	88:
		BCGapMove:=FALSE;
		BCGapState:=0;
		BCGapBusy:=FALSE;
		BCGapDone:=TRUE;
		Error:=FALSE;
		ErrorID:=0;
		LeftTop_MC_MoveAbsolute.Execute:=FALSE;
		LeftBottom_MC_MoveAbsolute.Execute:=FALSE;
		RightTopLin_MC_MoveAbsolute.Execute:=FALSE;
		RightBottomLin_MC_MoveAbsolute.Execute:=FALSE;
		LeftIn_MC_MoveAbsolute.Execute:=FALSE;
		LeftOut_MC_MoveAbsolute.Execute:=FALSE;
		RightInLin_MC_MoveAbsolute.Execute:=FALSE;
		RightOutLin_MC_MoveAbsolute.Execute:=FALSE;
		fb_ton_BC.IN:=FALSE;
	89:
		BCGapMove:=FALSE;
		BCGapState:=0;
		BCGapBusy:=FALSE;
		BCGapDone:=FALSE;
		Error:=FALSE;
		ErrorID:=0;
		LeftTop_MC_MoveAbsolute.Execute:=FALSE;
		LeftBottom_MC_MoveAbsolute.Execute:=FALSE;
		RightTopLin_MC_MoveAbsolute.Execute:=FALSE;
		RightBottomLin_MC_MoveAbsolute.Execute:=FALSE;
		LeftIn_MC_MoveAbsolute.Execute:=FALSE;
		LeftOut_MC_MoveAbsolute.Execute:=FALSE;
		RightInLin_MC_MoveAbsolute.Execute:=FALSE;
		RightOutLin_MC_MoveAbsolute.Execute:=FALSE;
		fb_ton_BC.IN:=FALSE;
	99:
		BCGapMove:=FALSE;
		BCGapState:=99;
		BCGapBusy:=FALSE;
		BCGapDone:=FALSE;
		Error:=TRUE;
		LeftTop_MC_MoveAbsolute.Execute:=FALSE;
		LeftBottom_MC_MoveAbsolute.Execute:=FALSE;
		RightTopLin_MC_MoveAbsolute.Execute:=FALSE;
		RightBottomLin_MC_MoveAbsolute.Execute:=FALSE;
		LeftIn_MC_MoveAbsolute.Execute:=FALSE;
		LeftOut_MC_MoveAbsolute.Execute:=FALSE;
		RightInLin_MC_MoveAbsolute.Execute:=FALSE;
		RightOutLin_MC_MoveAbsolute.Execute:=FALSE;
		fb_ton_BC.IN:=FALSE;
	-100:
		FB_PlcEmergencyStop();
		BCGapMove:=FALSE;
		BCGapState:=-100;
		BCGapBusy:=FALSE;
		BCGapDone:=FALSE;
		Error:=TRUE;
		LeftTop_MC_MoveAbsolute.Execute:=FALSE;
		LeftBottom_MC_MoveAbsolute.Execute:=FALSE;
		RightTopLin_MC_MoveAbsolute.Execute:=FALSE;
		RightBottomLin_MC_MoveAbsolute.Execute:=FALSE;
		LeftIn_MC_MoveAbsolute.Execute:=FALSE;
		LeftOut_MC_MoveAbsolute.Execute:=FALSE;
		RightInLin_MC_MoveAbsolute.Execute:=FALSE;
		RightOutLin_MC_MoveAbsolute.Execute:=FALSE;
		fb_ton_BC.IN:=FALSE;
END_CASE
END_IF
END_ACTION

ACTION A_BottomMove:
IF BottomMove THEN
BottomBusy:=TRUE;
BottomDone:=FALSE;
fb_ton2(PT:=t#80s);(*2mm/s max spees,120mmÐÐ³Ì£¬60sÄÚ×ßÍê*)
A_MoveMC();
CASE BottomState OF

	0:
		IF  LeftBottom_MC_MoveAbsolute.Error OR RightBottomLin_MC_MoveAbsolute.Error THEN		(*¼ì²éMC Error*)
			ErrorID:=2;
			BottomState:=99;
		END_IF
		BottomState:=1;

	1:
		LeftBottom_MC_MoveAbsolute.Position:=BottomPosition;
		LeftBottom_MC_MoveAbsolute.Velocity:=BottomVelocity;
		LeftBottom_MC_MoveAbsolute.Execute:=TRUE;
		RightBottomLin_MC_MoveAbsolute.Position:=BottomPosition;
		RightBottomLin_MC_MoveAbsolute.Velocity:=BottomVelocity;
		RightBottomLin_MC_MoveAbsolute.Execute:=TRUE;
		fb_ton2.IN:=TRUE;
		BottomState:=2;
	2:
		IF NOT LeftBottom_MC_MoveAbsolute.Done THEN		(*ÔË¶¯ÖÐ£¬¼ì²éDoneÐÅºÅ£¬Ã»ÓÐÔòÑ­»·£¬³¬Ê±±¨´í*)
			BottomState:=2;
		ELSIF LeftBottom_MC_MoveAbsolute.Done THEN		(*ÔË¶¯Íê³É£¬×ªÏÂÒ»²½*)
				BottomState:=88;
		END_IF
		(*½ÓÊÕµ½stopÐÅºÅÊ±£¬reset×´Ì¬*)
		IF BottomReset THEN
			BottomState:=89;
		END_IF

	88:
		BottomMove:=FALSE;
		BottomState:=0;
		BottomBusy:=FALSE;
		BottomDone:=TRUE;
		Error:=FALSE;
		ErrorID:=0;
		LeftBottom_MC_MoveAbsolute.Execute:=FALSE;
		RightBottomLin_MC_MoveAbsolute.Execute:=FALSE;
		fb_ton2.IN:=FALSE;
	89:
		BottomMove:=FALSE;
		BottomState:=0;
		BottomBusy:=FALSE;
		BottomDone:=FALSE;
		Error:=FALSE;
		ErrorID:=0;
		LeftBottom_MC_MoveAbsolute.Execute:=FALSE;
		RightBottomLin_MC_MoveAbsolute.Execute:=FALSE;
		fb_ton2.IN:=FALSE;
	99:
		BottomMove:=FALSE;
		BottomState:=99;
		BottomBusy:=FALSE;
		BottomDone:=FALSE;
		Error:=TRUE;
		LeftBottom_MC_MoveAbsolute.Execute:=FALSE;
		RightBottomLin_MC_MoveAbsolute.Execute:=FALSE;
		fb_ton2.IN:=FALSE;
	-100:
		FB_PlcEmergencyStop();
		BottomMove:=FALSE;
		BottomState:=-100;
		BottomBusy:=FALSE;
		BottomDone:=FALSE;
		Error:=TRUE;
		LeftBottom_MC_MoveAbsolute.Execute:=FALSE;
		RightBottomLin_MC_MoveAbsolute.Execute:=FALSE;
		fb_ton2.IN:=FALSE;
END_CASE
END_IF
END_ACTION

ACTION A_InMove:
IF InMove THEN
InBusy:=TRUE;
InDone:=FALSE;
fb_ton3(PT:=T#80S);(*2mm/s max spees,120mmÐÐ³Ì£¬60sÄÚ×ßÍê*)
A_MoveMC();
CASE InState OF
	0:
		IF LeftIn_MC_MoveAbsolute.Error OR RightInLin_MC_MoveAbsolute.Error THEN		(*¼ì²éMC Error*)
			ErrorID:=2;
			InState:=99;
		END_IF
		InState:=1;
	1:
		LeftIn_MC_MoveAbsolute.Position:=InPosition;
		LeftIn_MC_MoveAbsolute.Velocity:=InVelocity;
		LeftIn_MC_MoveAbsolute.Execute:=TRUE;
		RightInLin_MC_MoveAbsolute.Position:=InPosition;
		RightInLin_MC_MoveAbsolute.Velocity:=InVelocity;
		RightInLin_MC_MoveAbsolute.Execute:=TRUE;
		fb_ton3.IN:=TRUE;
		InState:=2;
	2:
		IF NOT LeftIn_MC_MoveAbsolute.Done OR NOT RightInLin_MC_MoveAbsolute.Done THEN		(*ÔË¶¯ÖÐ£¬¼ì²éDoneÐÅºÅ£¬Ã»ÓÐÔòÑ­»·£¬³¬Ê±±¨´í*)
			InState:=2;
		ELSIF LeftIn_MC_MoveAbsolute.Done AND RightInLin_MC_MoveAbsolute.Done THEN		(*ÔË¶¯Íê³É£¬×ªÏÂÒ»²½*)
				InState:=88;
		END_IF
		(*½ÓÊÕµ½sInÐÅºÅÊ±£¬reset×´Ì¬*)
		IF InReset THEN
			InState:=89;
		END_IF

	88:
		InMove:=FALSE;
		InState:=0;
		InBusy:=FALSE;
		InDone:=TRUE;
		Error:=FALSE;
		ErrorID:=0;
		LeftIn_MC_MoveAbsolute.Execute:=FALSE;
		RightInLin_MC_MoveAbsolute.Execute:=FALSE;
		fb_ton3.IN:=FALSE;
	89:
		InMove:=FALSE;
		InState:=0;
		InBusy:=FALSE;
		InDone:=FALSE;
		Error:=FALSE;
		ErrorID:=0;
		LeftIn_MC_MoveAbsolute.Execute:=FALSE;
		RightInLin_MC_MoveAbsolute.Execute:=FALSE;
		fb_ton3.IN:=FALSE;
	99:
		InMove:=FALSE;
		InState:=99;
		InBusy:=FALSE;
		InDone:=FALSE;
		Error:=TRUE;
		LeftIn_MC_MoveAbsolute.Execute:=FALSE;
		RightInLin_MC_MoveAbsolute.Execute:=FALSE;
		fb_ton3.IN:=FALSE;
	-100:
		FB_PlcEmergencyStop();
		InMove:=FALSE;
		InState:=-100;
		InBusy:=FALSE;
		InDone:=FALSE;
		Error:=TRUE;
		LeftIn_MC_MoveAbsolute.Execute:=FALSE;
		RightInLin_MC_MoveAbsolute.Execute:=FALSE;
		fb_ton3.IN:=FALSE;
END_CASE
END_IF
END_ACTION

ACTION A_LeftBottomMove:
IF LeftBottomMove THEN
LeftBottomBusy:=TRUE;
LeftBottomDone:=FALSE;
fb_ton_debug_3(PT:=t#10s);

A_MoveMC();
CASE LeftBottomState OF
	0:
		IF LeftBottom_MC_MoveAbsolute.Error THEN		(*¼ì²éMC Error*)
			ErrorID:=2;
			LeftBottomState:=99;
		ELSIF leftBottomLin.Status.NotMoving THEN	(*Öá¶¼´¦ÓÚÍ£Ö¹×´Ì¬Ê±£¬×ªÏÂÒ»²½*)
			LeftBottomState:=1;
		END_IF
	1:
		LeftBottom_MC_MoveAbsolute.Position:=LeftBottomPosition;
		LeftBottom_MC_MoveAbsolute.Velocity:=LeftBottomVelocity;
		LeftBottom_MC_MoveAbsolute.Execute:=TRUE;
		fb_ton_debug_3.IN:=TRUE;
		LeftBottomState:=2;
	2:
		IF NOT LeftBottom_MC_MoveAbsolute.Done THEN		(*ÔË¶¯ÖÐ£¬¼ì²éDoneÐÅºÅ£¬Ã»ÓÐÔòÑ­»·£¬³¬Ê±±¨´í*)
			LeftBottomState:=2;
		ELSIF LeftBottom_MC_MoveAbsolute.Done THEN		(*ÔË¶¯Íê³É£¬×ªÏÂÒ»²½*)
				LeftBottomState:=88;
		END_IF
		(*½ÓÊÕµ½stopÐÅºÅÊ±£¬reset×´Ì¬*)
		IF LeftBottomReset THEN
			LeftBottomState:=89;
		END_IF

	88:
		LeftBottomMove:=FALSE;
		LeftBottomState:=0;
		LeftBottomBusy:=FALSE;
		LeftBottomDone:=TRUE;
		Error:=FALSE;
		ErrorID:=0;
		LeftBottom_MC_MoveAbsolute.Execute:=FALSE;
		fb_ton_debug_3.IN:=FALSE;
	89:
		LeftBottomMove:=FALSE;
		LeftBottomState:=0;
		LeftBottomBusy:=FALSE;
		LeftBottomDone:=FALSE;
		Error:=FALSE;
		ErrorID:=0;
		LeftBottom_MC_MoveAbsolute.Execute:=FALSE;
		fb_ton_debug_3.IN:=FALSE;
	99:
		LeftBottomMove:=FALSE;
		LeftBottomState:=99;
		LeftBottomBusy:=FALSE;
		LeftBottomDone:=FALSE;
		Error:=TRUE;
		LeftBottom_MC_MoveAbsolute.Execute:=FALSE;
		fb_ton_debug_3.IN:=FALSE;
	-100:
		FB_PlcEmergencyStop();
		LeftBottomMove:=FALSE;
		LeftBottomState:=-100;
		LeftBottomBusy:=FALSE;
		LeftBottomDone:=FALSE;
		Error:=TRUE;
		LeftBottom_MC_MoveAbsolute.Execute:=FALSE;
		fb_ton_debug_3.IN:=FALSE;
END_CASE
END_IF
END_ACTION

ACTION A_LeftInMove:
IF LeftInMove THEN
LeftInBusy:=TRUE;
LeftInDone:=FALSE;
fb_ton_debug_5(PT:=T#10S);

A_MoveMC();
CASE LeftInState OF
	0:
		IF LeftIn_MC_MoveAbsolute.Error THEN		(*¼ì²éMC Error*)
			ErrorID:=2;
			LeftInState:=99;
		ELSIF leftInLin.Status.NotMoving THEN	(*Öá¶¼´¦ÓÚÍ£Ö¹×´Ì¬Ê±£¬×ªÏÂÒ»²½*)
			LeftInState:=1;
		END_IF
	1:
		LeftIn_MC_MoveAbsolute.Position:=LeftInPosition;
		LeftIn_MC_MoveAbsolute.Velocity:=LeftInVelocity;
		LeftIn_MC_MoveAbsolute.Execute:=TRUE;
		fb_ton_debug_5.IN:=TRUE;
		LeftInState:=2;
	2:
		IF NOT LeftIn_MC_MoveAbsolute.Done THEN		(*ÔË¶¯ÖÐ£¬¼ì²éDoneÐÅºÅ£¬Ã»ÓÐÔòÑ­»·£¬³¬Ê±±¨´í*)
			LeftInState:=2;
		ELSIF LeftIn_MC_MoveAbsolute.Done THEN		(*ÔË¶¯Íê³É£¬×ªÏÂÒ»²½*)
				LeftInState:=88;
		END_IF
		(*½ÓÊÕµ½stopÐÅºÅÊ±£¬reset×´Ì¬*)
		IF LeftInReset THEN
			LeftInState:=89;
		END_IF

	88:
		LeftInMove:=FALSE;
		LeftInState:=0;
		LeftInBusy:=FALSE;
		LeftInDone:=TRUE;
		Error:=FALSE;
		ErrorID:=0;
		LeftIn_MC_MoveAbsolute.Execute:=FALSE;
		fb_ton_debug_5.IN:=FALSE;
	89:
		LeftInMove:=FALSE;
		LeftInState:=0;
		LeftInBusy:=FALSE;
		LeftInDone:=FALSE;
		Error:=FALSE;
		ErrorID:=0;
		LeftIn_MC_MoveAbsolute.Execute:=FALSE;
		fb_ton_debug_5.IN:=FALSE;
	99:
		LeftInMove:=FALSE;
		LeftInState:=99;
		LeftInBusy:=FALSE;
		LeftInDone:=FALSE;
		Error:=TRUE;
		LeftIn_MC_MoveAbsolute.Execute:=FALSE;
		fb_ton_debug_5.IN:=FALSE;
	-100:
		FB_PlcEmergencyStop();
		LeftInMove:=FALSE;
		LeftInState:=-100;
		LeftInBusy:=FALSE;
		LeftInDone:=FALSE;
		Error:=TRUE;
		LeftIn_MC_MoveAbsolute.Execute:=FALSE;
		fb_ton_debug_5.IN:=FALSE;
END_CASE
END_IF
END_ACTION

ACTION A_LeftOutMove:
IF LeftOutMove THEN
LeftOutBusy:=TRUE;
LeftOutDone:=FALSE;
fb_ton_debug_7(PT:=t#10s);

A_MoveMC();
CASE LeftOutState OF
	0:
		IF LeftOut_MC_MoveAbsolute.Error THEN		(*¼ì²éMC Error*)
			ErrorID:=2;
			LeftOutState:=99;
		ELSIF leftOutLin.Status.NotMoving THEN	(*Öá¶¼´¦ÓÚÍ£Ö¹×´Ì¬Ê±£¬×ªÏÂÒ»²½*)
			LeftOutState:=1;
		END_IF
	1:
		LeftOut_MC_MoveAbsolute.Position:=LeftOutPosition;
		LeftOut_MC_MoveAbsolute.Velocity:=LeftOutVelocity;
		LeftOut_MC_MoveAbsolute.Execute:=TRUE;
		fb_ton_debug_7.IN:=TRUE;
		LeftOutState:=2;
	2:
		IF NOT LeftOut_MC_MoveAbsolute.Done THEN		(*ÔË¶¯ÖÐ£¬¼ì²éDoneÐÅºÅ£¬Ã»ÓÐÔòÑ­»·£¬³¬Ê±±¨´í*)
			LeftOutState:=2;
		ELSIF LeftOut_MC_MoveAbsolute.Done THEN		(*ÔË¶¯Íê³É£¬×ªÏÂÒ»²½*)
				LeftOutState:=88;
		END_IF
		(*½ÓÊÕµ½stopÐÅºÅÊ±£¬reset×´Ì¬*)
		IF LeftOutReset THEN
			LeftOutState:=89;
		END_IF

	88:
		LeftOutMove:=FALSE;
		LeftOutState:=0;
		LeftOutBusy:=FALSE;
		LeftOutDone:=TRUE;
		Error:=FALSE;
		ErrorID:=0;
		LeftOut_MC_MoveAbsolute.Execute:=FALSE;
		fb_ton_debug_7.IN:=FALSE;
	89:
		LeftOutMove:=FALSE;
		LeftOutState:=0;
		LeftOutBusy:=FALSE;
		LeftOutDone:=FALSE;
		Error:=FALSE;
		ErrorID:=0;
		LeftOut_MC_MoveAbsolute.Execute:=FALSE;
		fb_ton_debug_7.IN:=FALSE;
	99:
		LeftOutMove:=FALSE;
		LeftOutState:=99;
		LeftOutBusy:=FALSE;
		LeftOutDone:=FALSE;
		Error:=TRUE;
		LeftOut_MC_MoveAbsolute.Execute:=FALSE;
		fb_ton_debug_7.IN:=FALSE;
	-100:
		FB_PlcEmergencyStop();
		LeftOutMove:=FALSE;
		LeftOutState:=-100;
		LeftOutBusy:=FALSE;
		LeftOutDone:=FALSE;
		Error:=TRUE;
		LeftOut_MC_MoveAbsolute.Execute:=FALSE;
		fb_ton_debug_7.IN:=FALSE;
END_CASE
END_IF
END_ACTION

ACTION A_LeftTopMove:
IF LeftTopMove THEN
LeftTopBusy:=TRUE;
LeftTopDone:=FALSE;
fb_ton_debug_1(PT:=t#10s);

A_MoveMC();
CASE LeftTopState OF
	0:
		IF LeftTop_MC_MoveAbsolute.Error THEN		(*¼ì²éMC Error*)
			ErrorID:=2;
			LeftTopState:=99;
		ELSIF leftTopLin.Status.NotMoving THEN	(*Öá¶¼´¦ÓÚÍ£Ö¹×´Ì¬Ê±£¬×ªÏÂÒ»²½*)
			LeftTopState:=1;
		END_IF
	1:
		LeftTop_MC_MoveAbsolute.Position:=LeftTopPosition;
		LeftTop_MC_MoveAbsolute.Velocity:=LeftTopVelocity;
		LeftTop_MC_MoveAbsolute.Execute:=TRUE;
		fb_ton_debug_1.IN:=TRUE;
		LeftTopState:=2;
	2:
		IF NOT LeftTop_MC_MoveAbsolute.Done THEN		(*ÔË¶¯ÖÐ£¬¼ì²éDoneÐÅºÅ£¬Ã»ÓÐÔòÑ­»·£¬³¬Ê±±¨´í*)
			LeftTopState:=2;
		ELSIF LeftTop_MC_MoveAbsolute.Done THEN		(*ÔË¶¯Íê³É£¬×ªÏÂÒ»²½*)
				LeftTopState:=88;
		END_IF
		(*½ÓÊÕµ½stopÐÅºÅÊ±£¬reset×´Ì¬*)
		IF LeftTopReset THEN
			LeftTopState:=89;
		END_IF

	88:
		LeftTopMove:=FALSE;
		LeftTopState:=0;
		LeftTopBusy:=FALSE;
		LeftTopDone:=TRUE;
		Error:=FALSE;
		ErrorID:=0;
		LeftTop_MC_MoveAbsolute.Execute:=FALSE;
		fb_ton_debug_1.IN:=FALSE;
	89:
		LeftTopMove:=FALSE;
		LeftTopState:=0;
		LeftTopBusy:=FALSE;
		LeftTopDone:=FALSE;
		Error:=FALSE;
		ErrorID:=0;
		LeftTop_MC_MoveAbsolute.Execute:=FALSE;
		fb_ton_debug_1.IN:=FALSE;
	99:
		LeftTopMove:=FALSE;
		LeftTopState:=99;
		LeftTopBusy:=FALSE;
		LeftTopDone:=FALSE;
		Error:=TRUE;
		LeftTop_MC_MoveAbsolute.Execute:=FALSE;
		fb_ton_debug_1.IN:=FALSE;
	-100:
		FB_PlcEmergencyStop();
		LeftTopMove:=FALSE;
		LeftTopState:=-100;
		LeftTopBusy:=FALSE;
		LeftTopDone:=FALSE;
		Error:=TRUE;
		LeftTop_MC_MoveAbsolute.Execute:=FALSE;
		fb_ton_debug_1.IN:=FALSE;
END_CASE
END_IF
END_ACTION

ACTION A_MoveMC:
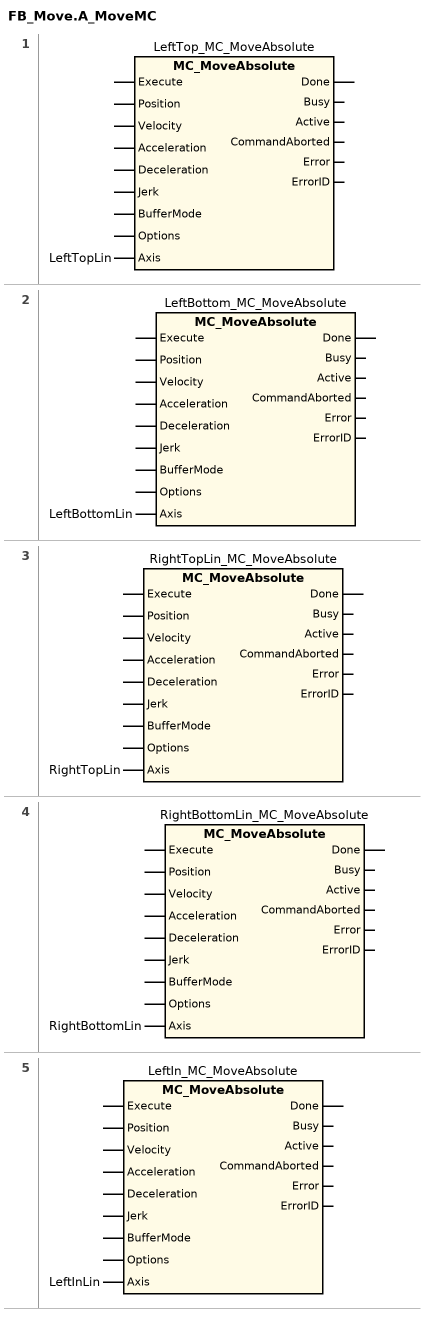
// NETWORK 1
LeftTop_MC_MoveAbsolute(Axis := LeftTopLin); // MC_MoveAbsolute

// NETWORK 2
LeftBottom_MC_MoveAbsolute(Axis := LeftBottomLin); // MC_MoveAbsolute

// NETWORK 3
RightTopLin_MC_MoveAbsolute(Axis := RightTopLin); // MC_MoveAbsolute

// NETWORK 4
RightBottomLin_MC_MoveAbsolute(Axis := RightBottomLin); // MC_MoveAbsolute

// NETWORK 5
LeftIn_MC_MoveAbsolute(Axis := LeftInLin); // MC_MoveAbsolute

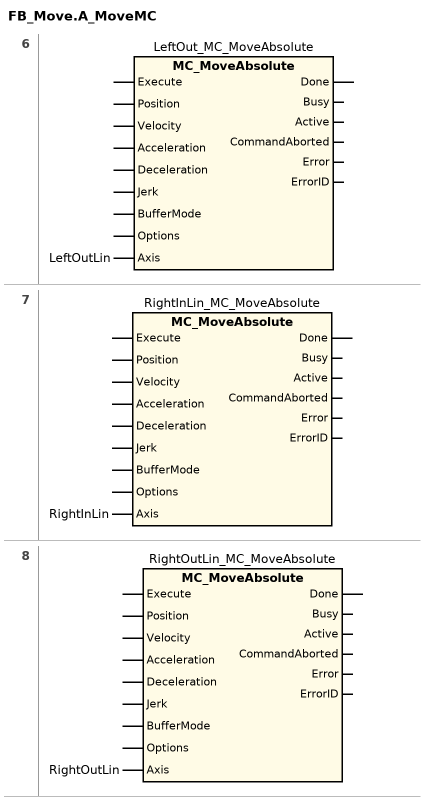
// NETWORK 6
LeftOut_MC_MoveAbsolute(Axis := LeftOutLin); // MC_MoveAbsolute

// NETWORK 7
RightInLin_MC_MoveAbsolute(Axis := RightInLin); // MC_MoveAbsolute

// NETWORK 8
RightOutLin_MC_MoveAbsolute(Axis := RightOutLin); // MC_MoveAbsolute
END_ACTION

ACTION A_OutMove:
IF OutMove THEN
OutBusy:=TRUE;
OutDone:=FALSE;
fb_ton4(PT:=T#80S);(*2mm/s max spees,120mmÐÐ³Ì£¬60sÄÚ×ßÍê*)
A_MoveMC();
CASE OutState OF

	0:
		IF  LeftOut_MC_MoveAbsolute.Error OR RightOutLin_MC_MoveAbsolute.Error THEN		(*¼ì²éMC Error*)
			ErrorID:=2;
			OutState:=99;
		END_IF
		OutState:=1;

	1:
		LeftOut_MC_MoveAbsolute.Position:=OutPosition;
		LeftOut_MC_MoveAbsolute.Velocity:=OutVelocity;
		LeftOut_MC_MoveAbsolute.Execute:=TRUE;
		RightOutLin_MC_MoveAbsolute.Position:=OutPosition;
		RightOutLin_MC_MoveAbsolute.Velocity:=OutVelocity;
		RightOutLin_MC_MoveAbsolute.Execute:=TRUE;
		fb_ton4.IN:=TRUE;
		OutState:=2;
	2:
		IF NOT LeftOut_MC_MoveAbsolute.Done THEN		(*ÔË¶¯ÖÐ£¬¼ì²éDoneÐÅºÅ£¬Ã»ÓÐÔòÑ­»·£¬³¬Ê±±¨´í*)
			OutState:=2;
		ELSIF LeftOut_MC_MoveAbsolute.Done THEN		(*ÔË¶¯Íê³É£¬×ªÏÂÒ»²½*)
				OutState:=88;
		END_IF
		(*½ÓÊÕµ½stopÐÅºÅÊ±£¬reset×´Ì¬*)
		IF OutReset THEN
			OutState:=89;
		END_IF

	88:
		OutMove:=FALSE;
		OutState:=0;
		OutBusy:=FALSE;
		OutDone:=TRUE;
		Error:=FALSE;
		ErrorID:=0;
		LeftOut_MC_MoveAbsolute.Execute:=FALSE;
		RightOutLin_MC_MoveAbsolute.Execute:=FALSE;
		fb_ton4.IN:=FALSE;
	89:
		OutMove:=FALSE;
		OutState:=0;
		OutBusy:=FALSE;
		OutDone:=FALSE;
		Error:=FALSE;
		ErrorID:=0;
		LeftOut_MC_MoveAbsolute.Execute:=FALSE;
		RightOutLin_MC_MoveAbsolute.Execute:=FALSE;
		fb_ton4.IN:=FALSE;
	99:
		OutMove:=FALSE;
		OutState:=99;
		OutBusy:=FALSE;
		OutDone:=FALSE;
		Error:=TRUE;
		LeftOut_MC_MoveAbsolute.Execute:=FALSE;
		RightOutLin_MC_MoveAbsolute.Execute:=FALSE;
		fb_ton4.IN:=FALSE;
	-100:
		FB_PlcEmergencyStop();
		OutMove:=FALSE;
		OutState:=-100;
		OutBusy:=FALSE;
		OutDone:=FALSE;
		Error:=TRUE;
		LeftOut_MC_MoveAbsolute.Execute:=FALSE;
		RightOutLin_MC_MoveAbsolute.Execute:=FALSE;
		fb_ton4.IN:=FALSE;
END_CASE
END_IF
END_ACTION

ACTION A_RightBottomMove:
IF RightBottomMove THEN
RightBottomBusy:=TRUE;
RightBottomDone:=FALSE;
fb_ton_debug_4(PT:=t#10s);

A_MoveMC();
CASE RightBottomState OF
	0:
		IF RightBottomLin_MC_MoveAbsolute.Error THEN		(*¼ì²éMC Error*)
			ErrorID:=2;
			RightBottomState:=99;
		ELSIF RightBottomLin.Status.NotMoving THEN	(*Öá¶¼´¦ÓÚÍ£Ö¹×´Ì¬Ê±£¬×ªÏÂÒ»²½*)
			RightBottomState:=1;
		END_IF
	1:
		RightBottomLin_MC_MoveAbsolute.Position:=RightBottomPosition;
		RightBottomLin_MC_MoveAbsolute.Velocity:=RightBottomVelocity;
		RightBottomLin_MC_MoveAbsolute.Execute:=TRUE;
		fb_ton_debug_4.IN:=TRUE;
		RightBottomState:=2;
	2:
		IF NOT RightBottomLin_MC_MoveAbsolute.Done THEN		(*ÔË¶¯ÖÐ£¬¼ì²éDoneÐÅºÅ£¬Ã»ÓÐÔòÑ­»·£¬³¬Ê±±¨´í*)
			RightBottomState:=2;
		ELSIF RightBottomLin_MC_MoveAbsolute.Done THEN		(*ÔË¶¯Íê³É£¬×ªÏÂÒ»²½*)
				RightBottomState:=88;
		END_IF
		(*½ÓÊÕµ½stopÐÅºÅÊ±£¬reset×´Ì¬*)
		IF RightBottomReset THEN
			RightBottomState:=89;
		END_IF

	88:
		RightBottomMove:=FALSE;
		RightBottomState:=0;
		RightBottomBusy:=FALSE;
		RightBottomDone:=TRUE;
		Error:=FALSE;
		ErrorID:=0;
		RightBottomLin_MC_MoveAbsolute.Execute:=FALSE;
		fb_ton_debug_4.IN:=FALSE;
	89:
		RightBottomMove:=FALSE;
		RightBottomState:=0;
		RightBottomBusy:=FALSE;
		RightBottomDone:=FALSE;
		Error:=FALSE;
		ErrorID:=0;
		RightBottomLin_MC_MoveAbsolute.Execute:=FALSE;
		fb_ton_debug_4.IN:=FALSE;
	99:
		RightBottomMove:=FALSE;
		RightBottomState:=99;
		RightBottomBusy:=FALSE;
		RightBottomDone:=FALSE;
		Error:=TRUE;
		RightBottomLin_MC_MoveAbsolute.Execute:=FALSE;
		fb_ton_debug_4.IN:=FALSE;
	-100:
		FB_PlcEmergencyStop();
		RightBottomMove:=FALSE;
		RightBottomState:=-100;
		RightBottomBusy:=FALSE;
		RightBottomDone:=FALSE;
		Error:=TRUE;
		RightBottomLin_MC_MoveAbsolute.Execute:=FALSE;
		fb_ton_debug_4.IN:=FALSE;
END_CASE
END_IF
END_ACTION

ACTION A_RightInMove:
IF RightInMove THEN
RightInBusy:=TRUE;
RightInDone:=FALSE;
fb_ton_debug_6(PT:=T#10S);

A_MoveMC();
CASE RightInState OF
	0:
		IF RightInLin_MC_MoveAbsolute.Error THEN		(*¼ì²éMC Error*)
			ErrorID:=2;
			RightInState:=99;
		ELSIF RightInLin.Status.NotMoving THEN	(*Öá¶¼´¦ÓÚÍ£Ö¹×´Ì¬Ê±£¬×ªÏÂÒ»²½*)
			RightInState:=1;
		END_IF
	1:
		RightInLin_MC_MoveAbsolute.Position:=RightInPosition;
		RightInLin_MC_MoveAbsolute.Velocity:=RightInVelocity;
		RightInLin_MC_MoveAbsolute.Execute:=TRUE;
		fb_ton_debug_6.IN:=TRUE;
		RightInState:=2;
	2:
		IF NOT RightInLin_MC_MoveAbsolute.Done THEN		(*ÔË¶¯ÖÐ£¬¼ì²éDoneÐÅºÅ£¬Ã»ÓÐÔòÑ­»·£¬³¬Ê±±¨´í*)
				RightInState:=2;
		ELSIF RightInLin_MC_MoveAbsolute.Done THEN		(*ÔË¶¯Íê³É£¬×ªÏÂÒ»²½*)
				RightInState:=88;
		END_IF
		(*½ÓÊÕµ½stopÐÅºÅÊ±£¬reset×´Ì¬*)
		IF RightInReset THEN
			RightInState:=89;
		END_IF

	88:
		RightInMove:=FALSE;
		RightInState:=0;
		RightInBusy:=FALSE;
		RightInDone:=TRUE;
		Error:=FALSE;
		ErrorID:=0;
		RightInLin_MC_MoveAbsolute.Execute:=FALSE;
		fb_ton_debug_6.IN:=FALSE;
	89:
		RightInMove:=FALSE;
		RightInState:=0;
		RightInBusy:=FALSE;
		RightInDone:=FALSE;
		Error:=FALSE;
		ErrorID:=0;
		RightInLin_MC_MoveAbsolute.Execute:=FALSE;
		fb_ton_debug_6.IN:=FALSE;
	99:
		RightInMove:=FALSE;
		RightInState:=99;
		RightInBusy:=FALSE;
		RightInDone:=FALSE;
		Error:=TRUE;
		RightInLin_MC_MoveAbsolute.Execute:=FALSE;
		fb_ton_debug_6.IN:=FALSE;
	-100:
		FB_PlcEmergencyStop();
		RightInMove:=FALSE;
		RightInState:=-100;
		RightInBusy:=FALSE;
		RightInDone:=FALSE;
		Error:=TRUE;
		RightInLin_MC_MoveAbsolute.Execute:=FALSE;
		fb_ton_debug_6.IN:=FALSE;
END_CASE
END_IF
END_ACTION

ACTION A_RightOutMove:
IF RightOutMove THEN
RightOutBusy:=TRUE;
RightOutDone:=FALSE;
fb_ton_debug_8(PT:=T#10S);

A_MoveMC();
CASE RightOutState OF
	0:
		IF RightOutLin_MC_MoveAbsolute.Error THEN		(*¼ì²éMC Error*)
			ErrorID:=2;
			RightOutState:=99;
		ELSIF RightOutLin.Status.NotMoving THEN	(*Öá¶¼´¦ÓÚÍ£Ö¹×´Ì¬Ê±£¬×ªÏÂÒ»²½*)
			RightOutState:=1;
		END_IF
	1:
		RightOutLin_MC_MoveAbsolute.Position:=RightOutPosition;
		RightOutLin_MC_MoveAbsolute.Velocity:=RightOutVelocity;
		RightOutLin_MC_MoveAbsolute.Execute:=TRUE;
		fb_ton_debug_8.IN:=TRUE;
		RightOutState:=2;
	2:
		IF NOT RightOutLin_MC_MoveAbsolute.Done THEN		(*ÔË¶¯ÖÐ£¬¼ì²éDoneÐÅºÅ£¬Ã»ÓÐÔòÑ­»·£¬³¬Ê±±¨´í*)
			RightOutState:=2;
		ELSIF RightOutLin_MC_MoveAbsolute.Done THEN		(*ÔË¶¯Íê³É£¬×ªÏÂÒ»²½*)
				RightOutState:=88;
		END_IF
		(*½ÓÊÕµ½stopÐÅºÅÊ±£¬reset×´Ì¬*)
		IF RightOutReset THEN
			RightOutState:=89;
		END_IF

	88:
		RightOutMove:=FALSE;
		RightOutState:=0;
		RightOutBusy:=FALSE;
		RightOutDone:=TRUE;
		Error:=FALSE;
		ErrorID:=0;
		RightOutLin_MC_MoveAbsolute.Execute:=FALSE;
		fb_ton_debug_8.IN:=FALSE;
	89:
		RightOutMove:=FALSE;
		RightOutState:=0;
		RightOutBusy:=FALSE;
		RightOutDone:=FALSE;
		Error:=FALSE;
		ErrorID:=0;
		RightOutLin_MC_MoveAbsolute.Execute:=FALSE;
		fb_ton_debug_8.IN:=FALSE;
	99:
		RightOutMove:=FALSE;
		RightOutState:=99;
		RightOutBusy:=FALSE;
		RightOutDone:=FALSE;
		Error:=TRUE;
		RightOutLin_MC_MoveAbsolute.Execute:=FALSE;
		fb_ton_debug_8.IN:=FALSE;
	-100:
		FB_PlcEmergencyStop();
		RightOutMove:=FALSE;
		RightOutState:=-100;
		RightOutBusy:=FALSE;
		RightOutDone:=FALSE;
		Error:=TRUE;
		RightOutLin_MC_MoveAbsolute.Execute:=FALSE;
		fb_ton_debug_8.IN:=FALSE;
END_CASE
END_IF
END_ACTION

ACTION A_RightTopMove:
IF RightTopMove THEN
RightTopBusy:=TRUE;
RightTopDone:=FALSE;
fb_ton_debug_2(PT:=t#10s);

A_MoveMC();
CASE RightTopState OF
	0:
		IF RightTopLin_MC_MoveAbsolute.Error THEN		(*¼ì²éMC Error*)
			ErrorID:=2;
			RightTopState:=99;
		ELSIF RightTopLin.Status.NotMoving THEN	(*Öá¶¼´¦ÓÚÍ£Ö¹×´Ì¬Ê±£¬×ªÏÂÒ»²½*)
			RightTopState:=1;
		END_IF
	1:
		RightTopLin_MC_MoveAbsolute.Position:=RightTopPosition;
		RightTopLin_MC_MoveAbsolute.Velocity:=RightTopVelocity;
		RightTopLin_MC_MoveAbsolute.Execute:=TRUE;
		fb_ton_debug_2.IN:=TRUE;
		RightTopState:=2;
	2:
		IF NOT RightTopLin_MC_MoveAbsolute.Done THEN		(*ÔË¶¯ÖÐ£¬¼ì²éDoneÐÅºÅ£¬Ã»ÓÐÔòÑ­»·£¬³¬Ê±±¨´í*)
			RightTopState:=2;
		ELSIF RightTopLin_MC_MoveAbsolute.Done THEN		(*ÔË¶¯Íê³É£¬×ªÏÂÒ»²½*)
				RightTopState:=88;
		END_IF
		(*½ÓÊÕµ½stopÐÅºÅÊ±£¬reset×´Ì¬*)
		IF RightTopReset THEN
			RightTopState:=89;
		END_IF

	88:
		RightTopMove:=FALSE;
		RightTopState:=0;
		RightTopBusy:=FALSE;
		RightTopDone:=TRUE;
		Error:=FALSE;
		ErrorID:=0;
		RightTopLin_MC_MoveAbsolute.Execute:=FALSE;
		fb_ton_debug_2.IN:=FALSE;
	89:
		RightTopMove:=FALSE;
		RightTopState:=0;
		RightTopBusy:=FALSE;
		RightTopDone:=FALSE;
		Error:=FALSE;
		ErrorID:=0;
		RightTopLin_MC_MoveAbsolute.Execute:=FALSE;
		fb_ton_debug_2.IN:=FALSE;
	99:
		RightTopMove:=FALSE;
		RightTopState:=99;
		RightTopBusy:=FALSE;
		RightTopDone:=FALSE;
		Error:=TRUE;
		RightTopLin_MC_MoveAbsolute.Execute:=FALSE;
		fb_ton_debug_2.IN:=FALSE;
	-100:
		FB_PlcEmergencyStop();
		RightTopMove:=FALSE;
		RightTopState:=-100;
		RightTopBusy:=FALSE;
		RightTopDone:=FALSE;
		Error:=TRUE;
		RightTopLin_MC_MoveAbsolute.Execute:=FALSE;
		fb_ton_debug_2.IN:=FALSE;
END_CASE
END_IF
END_ACTION

ACTION A_TopMove:
IF TopMove THEN
TopBusy:=TRUE;
TopDone:=FALSE;
fb_ton1(PT:=t#80s);(*2mm/s max spees,120mmÐÐ³Ì£¬60sÄÚ×ßÍê*)
A_MoveMC();
CASE TopState OF
	0:
		IF LeftTop_MC_MoveAbsolute.Error OR RightTopLin_MC_MoveAbsolute.Error THEN		(*¼ì²éMC Error*)
			ErrorID:=2;
			TopState:=99;
		END_IF
		TopState:=1;
	1:
		LeftTop_MC_MoveAbsolute.Position:=TopPosition;
		LeftTop_MC_MoveAbsolute.Velocity:=TopVelocity;
		LeftTop_MC_MoveAbsolute.Execute:=TRUE;
		RightTopLin_MC_MoveAbsolute.Position:=TopPosition;
		RightTopLin_MC_MoveAbsolute.Velocity:=TopVelocity;
		RightTopLin_MC_MoveAbsolute.Execute:=TRUE;
		fb_ton1.IN:=TRUE;
		TopState:=2;
	2:
		IF NOT LeftTop_MC_MoveAbsolute.Done OR NOT RightTopLin_MC_MoveAbsolute.Done THEN		(*ÔË¶¯ÖÐ£¬¼ì²éDoneÐÅºÅ£¬Ã»ÓÐÔòÑ­»·£¬³¬Ê±±¨´í*)
			TopState:=2;
		ELSIF LeftTop_MC_MoveAbsolute.Done AND RightTopLin_MC_MoveAbsolute.Done THEN		(*ÔË¶¯Íê³É£¬×ªÏÂÒ»²½*)
				TopState:=88;
		END_IF
		(*½ÓÊÕµ½stopÐÅºÅÊ±£¬reset×´Ì¬*)
		IF TopReset THEN
			TopState:=89;
		END_IF

	88:
		TopMove:=FALSE;
		TopState:=0;
		TopBusy:=FALSE;
		TopDone:=TRUE;
		Error:=FALSE;
		ErrorID:=0;
		LeftTop_MC_MoveAbsolute.Execute:=FALSE;
		RightTopLin_MC_MoveAbsolute.Execute:=FALSE;
		fb_ton1.IN:=FALSE;
	89:
		TopMove:=FALSE;
		TopState:=0;
		TopBusy:=FALSE;
		TopDone:=FALSE;
		Error:=FALSE;
		ErrorID:=0;
		LeftTop_MC_MoveAbsolute.Execute:=FALSE;
		RightTopLin_MC_MoveAbsolute.Execute:=FALSE;
		fb_ton1.IN:=FALSE;
	99:
		TopMove:=FALSE;
		TopState:=99;
		TopBusy:=FALSE;
		TopDone:=FALSE;
		Error:=TRUE;
		LeftTop_MC_MoveAbsolute.Execute:=FALSE;
		RightTopLin_MC_MoveAbsolute.Execute:=FALSE;
		fb_ton1.IN:=FALSE;
	-100:
		FB_PlcEmergencyStop();
		TopMove:=FALSE;
		TopState:=-100;
		TopBusy:=FALSE;
		TopDone:=FALSE;
		Error:=TRUE;
		LeftTop_MC_MoveAbsolute.Execute:=FALSE;
		RightTopLin_MC_MoveAbsolute.Execute:=FALSE;
		fb_ton1.IN:=FALSE;
END_CASE
END_IF
END_ACTION

END_FUNCTION_BLOCK

// ---- POUs/CommonFB/MainFB/FB_Power.TcPOU
(****************************************************************
NAME:			FB_PowerOn
DATA:			2017.2.16
VERSION:		1.0.0
DESCRIPTION:	FB_PowerOn
HISTORY:
				2017.2.16		NEW

***************************************************************)
FUNCTION_BLOCK FB_Power
VAR_INPUT
	On:BOOL;
	Off:BOOL;
	Check:BOOL;
END_VAR
VAR_OUTPUT
	FbID:DINT:=1001;
	OnState:DINT;
	OffState: INT;
	OnBusy:BOOL;
	OffBusy:BOOL;
	OnStatus:BOOL;
	OffStatus: BOOL;
	Error:BOOL;
	ErrorID:DINT;
	PowerState:BOOL;
END_VAR
VAR
	LeftTopLin_MC_Power: MC_Power;
	RightTopLin_MC_Power: MC_Power;
	LeftBottomLin_MC_Power: MC_Power;
	RightBottomLin_MC_Power: MC_Power;
	LeftInLin_MC_Power: MC_Power;
	RightInLin_MC_Power: MC_Power;
	LeftOutLin_MC_Power: MC_Power;
	RightOutLin_MC_Power: MC_Power;
	fb_ton:TON;
END_VAR

(*power on *)
IF On AND NOT Off THEN
	A_PowerOn();
(*Power Off *)
ELSIF Off AND NOT On THEN
	A_PowerOff();
END_IF
(*Check*)
IF Check THEN
	A_CheckPowerStatus();
END_IF

ACTION A_CheckPowerStatus:
A_PowerMC();
IF  LeftTopLin_MC_Power.Status AND RightTopLin_MC_Power.Status
		AND LeftBottomLin_MC_Power.Status AND RightBottomLin_MC_Power.Status
		AND LeftInLin_MC_Power.Status AND RightInLin_MC_Power.Status
		AND LeftOutLin_MC_Power.Status AND RightOutLin_MC_Power.Status THEN
	PowerState:=1;
ELSIF NOT LeftTopLin_MC_Power.Status AND NOT RightTopLin_MC_Power.Status
		AND NOT LeftBottomLin_MC_Power.Status AND NOT RightBottomLin_MC_Power.Status
		AND NOT LeftInLin_MC_Power.Status AND NOT RightInLin_MC_Power.Status
		AND NOT LeftOutLin_MC_Power.Status AND NOT RightOutLin_MC_Power.Status THEN
	PowerState:=0;
ELSE
	//PowerState:=-1;
	//Error:=TRUE;
	//ErrorID:=77;
	(*FB_PlcEmergencyStop();*)
END_IF
END_ACTION

ACTION A_PowerMC:
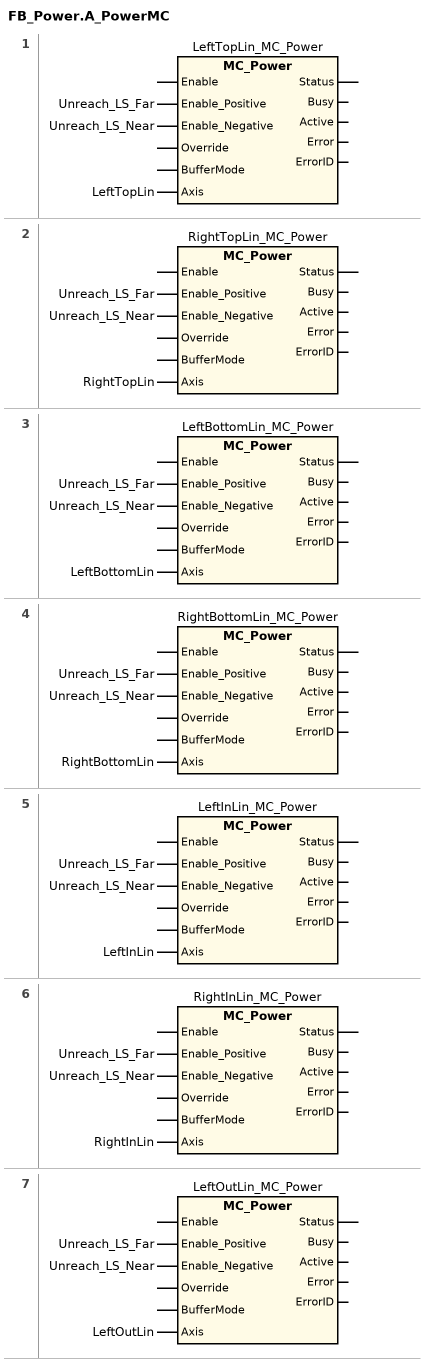
// NETWORK 1
LeftTopLin_MC_Power(
    Enable_Positive := Unreach_LS_Far,
    Enable_Negative := Unreach_LS_Near,
    Axis := LeftTopLin); // MC_Power

// NETWORK 2
RightTopLin_MC_Power(
    Enable_Positive := Unreach_LS_Far,
    Enable_Negative := Unreach_LS_Near,
    Axis := RightTopLin); // MC_Power

// NETWORK 3
LeftBottomLin_MC_Power(
    Enable_Positive := Unreach_LS_Far,
    Enable_Negative := Unreach_LS_Near,
    Axis := LeftBottomLin); // MC_Power

// NETWORK 4
RightBottomLin_MC_Power(
    Enable_Positive := Unreach_LS_Far,
    Enable_Negative := Unreach_LS_Near,
    Axis := RightBottomLin); // MC_Power

// NETWORK 5
LeftInLin_MC_Power(Enable_Positive := Unreach_LS_Far, Enable_Negative := Unreach_LS_Near, Axis := LeftInLin); // MC_Power

// NETWORK 6
RightInLin_MC_Power(
    Enable_Positive := Unreach_LS_Far,
    Enable_Negative := Unreach_LS_Near,
    Axis := RightInLin); // MC_Power

// NETWORK 7
LeftOutLin_MC_Power(
    Enable_Positive := Unreach_LS_Far,
    Enable_Negative := Unreach_LS_Near,
    Axis := LeftOutLin); // MC_Power

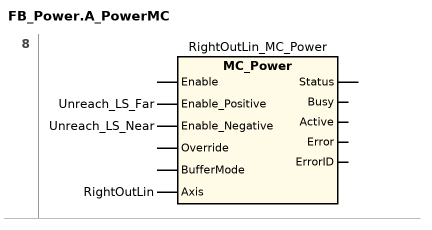
// NETWORK 8
RightOutLin_MC_Power(
    Enable_Positive := Unreach_LS_Far,
    Enable_Negative := Unreach_LS_Near,
    Axis := RightOutLin); // MC_Power
END_ACTION

ACTION A_PowerOff:
OffBusy:=TRUE;
CASE OffState OF
	0:
		IF NOT LeftTopLin_MC_Power.Status AND NOT RightTopLin_MC_Power.Status
			AND NOT LeftBottomLin_MC_Power.Status AND NOT RightBottomLin_MC_Power.Status
			AND NOT LeftInLin_MC_Power.Status AND NOT RightInLin_MC_Power.Status
			AND NOT LeftOutLin_MC_Power.Status AND NOT RightOutLin_MC_Power.Status THEN	(*¶¼Ã»ÉÏµç*)
			OffState:=88;
		ELSE
			OffState:=1;
		END_IF
	1:
		LeftTopLin_MC_Power.Enable:=FALSE;
		RightTopLin_MC_Power.Enable:=FALSE;
		LeftBottomLin_MC_Power.Enable:=FALSE;
		RightBottomLin_MC_Power.Enable:=FALSE;
		LeftInLin_MC_Power.Enable:=FALSE;
		RightInLin_MC_Power.Enable:=FALSE;
		LeftOutLin_MC_Power.Enable:=FALSE;
		RightOutLin_MC_Power.Enable:=FALSE;
		A_PowerMC();
		OffState:=2;
	2:
		IF NOT LeftTopLin_MC_Power.Status AND NOT RightTopLin_MC_Power.Status
			AND NOT LeftBottomLin_MC_Power.Status AND NOT RightBottomLin_MC_Power.Status
			AND NOT LeftInLin_MC_Power.Status AND NOT RightInLin_MC_Power.Status
			AND NOT LeftOutLin_MC_Power.Status AND NOT RightOutLin_MC_Power.Status THEN	(*¶¼Ã»ÉÏµç*)
			OffState:=88;
		ELSE
			ErrorId:=11;
			OffState:=-100;
		END_IF
	88:
		Off:=FALSE;
		OffState:=0;
		OffBusy:=FALSE;
		OnStatus:=FALSE;
		OffStatus:=TRUE;
		Error:=FALSE;
		ErrorID:=0;
	-100:
		FB_PlcEmergencyStop();
		Off:=FALSE;
		OffState:=-100;
		OffBusy:=FALSE;
		OffStatus:=FALSE;
		Error:=TRUE;

END_CASE
END_ACTION

ACTION A_PowerOn:
OnBusy:=TRUE;
fb_ton(PT:=t#0.5s);
CASE OnState OF
	0:	(*Check*)
		A_PowerMC();
		IF LeftTopLin_MC_Power.Error OR RightTopLin_MC_Power.Error
			OR LeftBottomLin_MC_Power.Error OR RightBottomLin_MC_Power.Error
			OR LeftInLin_MC_Power.Error OR RightInLin_MC_Power.Error
			OR LeftOutLin_MC_Power.Error OR RightOutLin_MC_Power.Error THEN	
			ErrorID:=1;
			OnState:=99;
		ELSIF LeftTopLin_MC_Power.Status OR RightTopLin_MC_Power.Status
			OR LeftBottomLin_MC_Power.Status OR RightBottomLin_MC_Power.Status 
			OR LeftInLin_MC_Power.Status OR RightInLin_MC_Power.Status
			OR LeftOutLin_MC_Power.Status OR RightOutLin_MC_Power.Status THEN		(*ÖáÒÑ¾­¶¼PowerOn£¬²»·ûºÏ¹¦ÄÜ¿éµ÷ÓÃÌõ¼þ*)
			ErrorID:=2;
			OnState:=-100;
		ELSIF NOT LeftTopLin_MC_Power.Status OR NOT RightTopLin_MC_Power.Status
			OR NOT LeftBottomLin_MC_Power.Status OR NOT RightBottomLin_MC_Power.Status 
			OR  NOT LeftInLin_MC_Power.Status OR NOT RightInLin_MC_Power.Status
			OR NOT LeftOutLin_MC_Power.Status OR NOT RightOutLin_MC_Power.Status THEN		(*Öá¶¼Ã»ÓÐPower£¬×ªÏÂÒ»²½*)
			OnState:=1;
		ELSE
			ErrorID:=3;
			OnState:=-100;
		END_IF
	1:	(*Execute*)
		IF NOT LeftTopLin_MC_Power.Status OR NOT RightTopLin_MC_Power.Status
			OR NOT LeftBottomLin_MC_Power.Status OR NOT RightBottomLin_MC_Power.Status
			OR NOT LeftInLin_MC_Power.Status OR NOT RightInLin_MC_Power.Status
			OR NOT LeftOutLin_MC_Power.Status OR NOT RightOutLin_MC_Power.Status THEN		(*ÔÙ¼ì²é£¬Öá¶¼Ã»ÓÐPower*)
			LeftTopLin_MC_Power.Enable:=TRUE;
			RightTopLin_MC_Power.Enable:=TRUE;
			LeftBottomLin_MC_Power.Enable:=TRUE;
			RightBottomLin_MC_Power.Enable:=TRUE;
			LeftInLin_MC_Power.Enable:=TRUE;
			RightInLin_MC_Power.Enable:=TRUE;
			LeftOutLin_MC_Power.Enable:=TRUE;
			RightOutLin_MC_Power.Enable:=TRUE;
			A_PowerMC();
			fb_ton.IN:=TRUE;
			OnState:=2;
		ELSE
			ErrorID:=4;
			OnState:=-100;
		END_IF
	2:	(*Wait*)
		A_PowerMC();
		IF NOT LeftTopLin_MC_Power.Status OR NOT RightTopLin_MC_Power.Status
			OR NOT LeftBottomLin_MC_Power.Status OR NOT RightBottomLin_MC_Power.Status
			OR NOT LeftInLin_MC_Power.Status OR NOT RightInLin_MC_Power.Status
			OR NOT LeftOutLin_MC_Power.Status OR NOT RightOutLin_MC_Power.Status THEN		(*Power StatusÐÅºÅ²»µ½£¬¼ÌÐøµÈ´ý£¬Èç¹û³¬Ê±ÔòFB Error*)
			IF NOT fb_ton.Q THEN
				OnState:=2;
			ELSE
				ErrorID:=8;
				OnState:=99;
			END_IF
		ELSIF  LeftTopLin_MC_Power.Status AND RightTopLin_MC_Power.Status
			AND LeftBottomLin_MC_Power.Status AND RightBottomLin_MC_Power.Status 
			AND   LeftInLin_MC_Power.Status AND RightInLin_MC_Power.Status
			AND LeftOutLin_MC_Power.Status AND RightOutLin_MC_Power.Status THEN			(*ÕýÈ·µç»úÉÏµã×´Ì¬£¬×ªÏÂÒ»²½*)
				OnState:=88;
		ELSE
				ErrorID:=9;
				OnState:=-100;
		END_IF
	88:
		On:=FALSE;
		OnState:=0;
		OnBusy:=FALSE;
		OnStatus:=TRUE;
		OffStatus:=FALSE;
		Error:=FALSE;
		ErrorID:=0;
		fb_ton.IN:=FALSE;
	99:
		On:=FALSE;
		OnState:=99;
		OnBusy:=FALSE;
		OnStatus:=FALSE;
		Error:=TRUE;
		LeftTopLin_MC_Power.Enable:=FALSE;
		RightTopLin_MC_Power.Enable:=FALSE;
		LeftBottomLin_MC_Power.Enable:=FALSE;
		RightBottomLin_MC_Power.Enable:=FALSE;
		LeftInLin_MC_Power.Enable:=FALSE;
		RightInLin_MC_Power.Enable:=FALSE;
		LeftOutLin_MC_Power.Enable:=FALSE;
		RightOutLin_MC_Power.Enable:=FALSE;
		fb_ton.IN:=FALSE;
	-100:
		FB_PlcEmergencyStop();
		On:=FALSE;
		OnState:=-100;
		OnBusy:=FALSE;
		OnStatus:=FALSE;
		Error:=TRUE;
		LeftTopLin_MC_Power.Enable:=FALSE;
		RightTopLin_MC_Power.Enable:=FALSE;
		LeftBottomLin_MC_Power.Enable:=FALSE;
		RightBottomLin_MC_Power.Enable:=FALSE;
		LeftInLin_MC_Power.Enable:=FALSE;
		RightInLin_MC_Power.Enable:=FALSE;
		LeftOutLin_MC_Power.Enable:=FALSE;
		RightOutLin_MC_Power.Enable:=FALSE;
		fb_ton.IN:=FALSE;

END_CASE
END_ACTION

END_FUNCTION_BLOCK

// ---- POUs/CommonFB/MainFB/FB_Stop.TcPOU
FUNCTION_BLOCK FB_Stop
VAR_INPUT
(*È«¾Ö*)
	Mode:DINT;
	PowerState:BOOL;
	CoupleState:DINT;
	(*GapMode*)
	GapStop:BOOL;
	(*BCGapMode*)
	BCGapStop:BOOL;
	(*SingleCarrierMode*)
	TopStop:BOOL;
	BottomStop:BOOL;
	InStop:BOOL;
	OutStop:BOOL;
	(*DebugMode*)
	LeftTopStop:BOOL;
	RightTopStop:BOOL;
	LeftBottomStop:BOOL;
	RightBottomStop:BOOL;
	LeftInStop:BOOL;
	RightInStop:BOOL;
	LeftOutStop:BOOL;
	RightOutStop:BOOL;
END_VAR
VAR_OUTPUT
	FbID:DINT:=1001;
	GapState:DINT;
	GapBusy:BOOL;
	GapDone:BOOL;

	BCGapState:DINT;
	BCGapBusy:BOOL;
	BCGapDone:BOOL;

	TopState:DINT;
	TopBusy:BOOL;
	TopDone:BOOL;
	BottomState:DINT;
	BottomBusy:BOOL;
	BottomDone:BOOL;
	InState:DINT;
	InBusy:BOOL;
	InDone:BOOL;
	OutState:DINT;
	OutBusy:BOOL;
	OutDone:BOOL;

	LeftTopState:DINT;
	LeftTopBusy:BOOL;
	LeftTopDone:BOOL;
	RightTopState:DINT;
	RightTopBusy:BOOL;
	RightTopDone:BOOL;
	LeftBottomState:DINT;
	LeftBottomBusy:BOOL;
	LeftBottomDone:BOOL;
	RightBottomState:DINT;
	RightBottomBusy:BOOL;
	RightBottomDone:BOOL;
	LeftInState:DINT;
	LeftInBusy:BOOL;
	LeftInDone:BOOL;
	RightInState:DINT;
	RightInBusy:BOOL;
	RightInDone:BOOL;
	LeftOutState:DINT;
	LeftOutBusy:BOOL;
	LeftOutDone:BOOL;
	RightOutState:DINT;
	RightOutBusy:BOOL;
	RightOutDone:BOOL;

	Error:BOOL;
	ErrorID:DINT;
END_VAR
VAR
	LeftTop_MC_Stop: MC_Stop;
	LeftBottom_MC_Stop: MC_Stop;
	RightTopLin_MC_Stop: MC_Stop;
	RightBottomLin_MC_Stop: MC_Stop;
	LeftIn_MC_Stop: MC_Stop;
	LeftOut_MC_Stop: MC_Stop;
	RightInLin_MC_Stop: MC_Stop;
	RightOutLin_MC_Stop: MC_Stop;
	fb_ton: TON;
	fb_ton1: TON;
	fb_ton2: TON;
	fb_ton3: TON;
	fb_ton4: TON;
	fb_ton_debug_1:TON;
	fb_ton_debug_2:TON;
	fb_ton_debug_3:TON;
	fb_ton_debug_4:TON;
	fb_ton_debug_5:TON;
	fb_ton_debug_6:TON;
	fb_ton_debug_7:TON;
	fb_ton_debug_8:TON;
	fb_ton_BC: TON;
END_VAR

IF PowerState=1 THEN
	IF Mode=1 AND TopStop THEN
		A_TopStop();
	ELSIF Mode=1 AND BottomStop THEN
		A_BottomStop();
	ELSIF Mode=1 AND InStop THEN
		A_InStop();
	ELSIF Mode=1 AND OutStop THEN
		A_OutStop();
	ELSIF Mode=2 AND LeftTopStop THEN
		A_LeftTopStop();
	ELSIF Mode=2 AND RightTopStop THEN
		A_RightTopStop();
	ELSIF Mode=2 AND LeftBottomStop THEN
		A_LeftBottomStop();
	ELSIF Mode=2 AND RightBottomStop THEN
		A_RightBottomStop();
	ELSIF Mode=2 AND LeftInStop THEN
		A_LeftInStop();
	ELSIF Mode=2 AND RightInStop THEN
		A_RightInStop();
	ELSIF Mode=2 AND LeftOutStop THEN
		A_LeftOutStop();
	ELSIF Mode=2 AND RightOutStop THEN
		A_RightOutStop();
	ELSIF Mode=5 AND BCGapStop THEN
		A_BCGapStop();
	ELSE
		FB_PlcEmergencyStop();
	END_IF
END_IF

ACTION A_BCGapStop:
IF BCGapStop THEN
BCGapBusy:=TRUE;
BCGapDone:=FALSE;
fb_ton_BC(PT:=t#100ms);
A_StopMC();
CASE BCGapState OF
	0:
		IF LeftTop_MC_Stop.Error OR LeftBottom_MC_Stop.Error 
			OR RightTopLin_MC_Stop.Error OR RightBottomLin_MC_Stop.Error
			OR  LeftIn_MC_Stop.Error OR LeftOut_MC_Stop.Error 
			OR RightInLin_MC_Stop.Error OR RightOutLin_MC_Stop.Error THEN
			ErrorID:=1;
			BCGapState:=-100;
			LeftTop_MC_Stop.Execute:=FALSE;
			LeftBottom_MC_Stop.Execute:=FALSE;
			RightTopLin_MC_Stop.Execute:=FALSE;
			RightBottomLin_MC_Stop.Execute:=FALSE;
			LeftIn_MC_Stop.Execute:=FALSE;
			LeftOut_MC_Stop.Execute:=FALSE;
			RightInLin_MC_Stop.Execute:=FALSE;
			RightOutLin_MC_Stop.Execute:=FALSE;
			A_StopMC();
		ELSE
			BCGapState:=1;
		END_IF
	1:
		LeftTop_MC_Stop.Execute:=TRUE;
		LeftBottom_MC_Stop.Execute:=TRUE;
		RightTopLin_MC_Stop.Execute:=TRUE;
		RightBottomLin_MC_Stop.Execute:=TRUE;
		LeftIn_MC_Stop.Execute:=TRUE;
		LeftOut_MC_Stop.Execute:=TRUE;
		RightInLin_MC_Stop.Execute:=TRUE;
		RightOutLin_MC_Stop.Execute:=TRUE;
		fb_ton_BC.IN:=TRUE;
		BCGapState:=2;
	2:
		IF  NOT LeftTop_MC_Stop.Done OR NOT LeftBottom_MC_Stop.Done 
			OR NOT RightTopLin_MC_Stop.Done OR NOT RightBottomLin_MC_Stop.Done
  			OR NOT LeftIn_MC_Stop.Done OR NOT LeftOut_MC_Stop.Done 
			OR NOT RightInLin_MC_Stop.Done OR NOT RightOutLin_MC_Stop.Done THEN
				BCGapState:=2;
		ELSE
			BCGapState:=88;
			LeftTop_MC_Stop.Execute:=FALSE;
			LeftBottom_MC_Stop.Execute:=FALSE;
			RightTopLin_MC_Stop.Execute:=FALSE;
			RightBottomLin_MC_Stop.Execute:=FALSE;			
			LeftIn_MC_Stop.Execute:=FALSE;
			LeftOut_MC_Stop.Execute:=FALSE;
			RightInLin_MC_Stop.Execute:=FALSE;
			RightOutLin_MC_Stop.Execute:=FALSE;
			A_StopMC();
		END_IF

	88:
		BCGapStop:=FALSE;
		BCGapState:=0;
		BCGapBusy:=FALSE;
		BCGapDone:=TRUE;
		Error:=FALSE;
		ErrorID:=0;
		fb_ton_BC.IN:=FALSE;

	-100:
		FB_PlcEmergencyStop();
		BCGapStop:=FALSE;
		BCGapState:=-100;
		BCGapBusy:=FALSE;
		BCGapDone:=FALSE;
		Error:=TRUE;
		LeftTop_MC_Stop.Execute:=FALSE;
		LeftBottom_MC_Stop.Execute:=FALSE;
		RightTopLin_MC_Stop.Execute:=FALSE;
		RightBottomLin_MC_Stop.Execute:=FALSE;			
		LeftIn_MC_Stop.Execute:=FALSE;
		LeftOut_MC_Stop.Execute:=FALSE;
		RightInLin_MC_Stop.Execute:=FALSE;
		RightOutLin_MC_Stop.Execute:=FALSE;
		A_StopMC();
		fb_ton_BC.IN:=FALSE;

END_CASE
END_IF
END_ACTION

ACTION A_BottomStop:
IF BottomStop THEN
BottomBusy:=TRUE;
BottomDone:=FALSE;
fb_ton2(PT:=t#100ms);
A_StopMC();
CASE BottomState OF
	0:
		IF LeftBottom_MC_Stop.Error OR RightBottomLin_MC_Stop.Error THEN
			ErrorID:=1;
			BottomState:=-100;
			LeftBottom_MC_Stop.Execute:=FALSE;
			RightBottomLin_MC_Stop.Execute:=FALSE;
			A_StopMC();
		ELSE
			BottomState:=1;
		END_IF
	1:
		LeftBottom_MC_Stop.Execute:=TRUE;
		RightBottomLin_MC_Stop.Execute:=TRUE;
		fb_ton2.IN:=TRUE;
		BottomState:=2;
	2:
		IF  NOT LeftBottom_MC_Stop.Done OR NOT LeftBottom_MC_Stop.Done THEN
				BottomState:=2;
		ELSE
			BottomState:=88;
			LeftBottom_MC_Stop.Execute:=FALSE;
			RightBottomLin_MC_Stop.Execute:=FALSE;
			A_StopMC();
		END_IF

	88:
		BottomStop:=FALSE;
		BottomState:=0;
		BottomBusy:=FALSE;
		BottomDone:=TRUE;
		Error:=FALSE;
		ErrorID:=0;
		fb_ton2.IN:=FALSE;

	-100:
		FB_PlcEmergencyStop();
		BottomStop:=FALSE;
		BottomState:=-100;
		BottomBusy:=FALSE;
		BottomDone:=FALSE;
		Error:=TRUE;
		LeftBottom_MC_Stop.Execute:=FALSE;
		RightBottomLin_MC_Stop.Execute:=FALSE;
		A_StopMC();
		fb_ton2.IN:=FALSE;

END_CASE
END_IF
END_ACTION

ACTION A_InStop:
IF InStop THEN
InBusy:=TRUE;
InDone:=FALSE;
fb_ton3(PT:=t#100ms);
A_StopMC();
CASE InState OF
	0:
		IF LeftIn_MC_Stop.Error OR RightInLin_MC_Stop.Error THEN
			ErrorID:=1;
			InState:=-100;
			LeftIn_MC_Stop.Execute:=FALSE;
			A_StopMC();
		ELSE
			InState:=1;
		END_IF
	1:
		LeftIn_MC_Stop.Execute:=TRUE;
		RightInLin_MC_Stop.Execute:=TRUE;
		fb_ton3.IN:=TRUE;
		InState:=2;
	2:
		IF  NOT LeftIn_MC_Stop.Done OR NOT RightInLin_MC_Stop.Done THEN
				InState:=2;
		ELSE
			InState:=88;
			LeftIn_MC_Stop.Execute:=FALSE;
			RightInLin_MC_Stop.Execute:=FALSE;
			A_StopMC();
		END_IF

	88:
		InStop:=FALSE;
		InState:=0;
		InBusy:=FALSE;
		InDone:=TRUE;
		Error:=FALSE;
		ErrorID:=0;
		fb_ton3.IN:=FALSE;

	-100:
		FB_PlcEmergencyStop();
		InStop:=FALSE;
		InState:=-100;
		InBusy:=FALSE;
		InDone:=FALSE;
		Error:=TRUE;
		LeftIn_MC_Stop.Execute:=FALSE;
		RightInLin_MC_Stop.Execute:=FALSE;
		A_StopMC();
		fb_ton3.IN:=FALSE;

END_CASE
END_IF
END_ACTION

ACTION A_LeftBottomStop:
IF LeftBottomStop THEN
LeftBottomBusy:=TRUE;
LeftBottomDone:=FALSE;
fb_ton_debug_3(PT:=t#100ms);
A_StopMC();
CASE LeftBottomState OF
	0:
		IF LeftBottom_MC_Stop.Error THEN
			ErrorID:=41;
			LeftBottomState:=-100;
			LeftBottom_MC_Stop.Execute:=FALSE;
			A_StopMC();
		ELSE
			LeftBottomState:=1;
		END_IF
	1:
		LeftBottom_MC_Stop.Execute:=TRUE;
		fb_ton_debug_3.IN:=TRUE;
		LeftBottomState:=2;
	2:
		IF  NOT LeftBottom_MC_Stop.Done THEN
				LeftBottomState:=2;
		ELSE
			LeftBottomState:=88;
			LeftBottom_MC_Stop.Execute:=FALSE;
			A_StopMC();
		END_IF

	88:
		LeftBottomStop:=FALSE;
		LeftBottomState:=0;
		LeftBottomBusy:=FALSE;
		LeftBottomDone:=TRUE;
		Error:=FALSE;
		ErrorID:=0;
		fb_ton_debug_3.IN:=FALSE;

	-100:
		FB_PlcEmergencyStop();
		LeftBottomStop:=FALSE;
		LeftBottomState:=-100;
		LeftBottomBusy:=FALSE;
		LeftBottomDone:=FALSE;
		Error:=TRUE;
		LeftBottom_MC_Stop.Execute:=FALSE;
		A_StopMC();
		fb_ton_debug_3.IN:=FALSE;

END_CASE
END_IF
END_ACTION

ACTION A_LeftInStop:
IF LeftInStop THEN
LeftInBusy:=TRUE;
LeftInDone:=FALSE;
fb_ton_debug_4(PT:=t#100ms);
A_StopMC();
CASE LeftInState OF
	0:
		IF LeftIn_MC_Stop.Error THEN
			ErrorID:=41;
			LeftInState:=-100;
			LeftIn_MC_Stop.Execute:=FALSE;
			A_StopMC();
		ELSE
			LeftInState:=1;
		END_IF
	1:
		LeftIn_MC_Stop.Execute:=TRUE;
		fb_ton_debug_4.IN:=TRUE;
		LeftInState:=2;
	2:
		IF  NOT LeftIn_MC_Stop.Done THEN
				LeftInState:=2;
		ELSE
			LeftInState:=88;
			LeftIn_MC_Stop.Execute:=FALSE;
			A_StopMC();
		END_IF

	88:
		LeftInStop:=FALSE;
		LeftInState:=0;
		LeftInBusy:=FALSE;
		LeftInDone:=TRUE;
		Error:=FALSE;
		ErrorID:=0;
		fb_ton_debug_4.IN:=FALSE;

	-100:
		FB_PlcEmergencyStop();
		LeftInStop:=FALSE;
		LeftInState:=-100;
		LeftInBusy:=FALSE;
		LeftInDone:=FALSE;
		Error:=TRUE;
		LeftIn_MC_Stop.Execute:=FALSE;
		A_StopMC();
		fb_ton_debug_4.IN:=FALSE;

END_CASE
END_IF
END_ACTION

ACTION A_LeftOutStop:
IF LeftOutStop THEN
LeftOutBusy:=TRUE;
LeftOutDone:=FALSE;
fb_ton_debug_7(PT:=t#100ms);
A_StopMC();
CASE LeftOutState OF
	0:
		IF LeftOut_MC_Stop.Error THEN
			ErrorID:=41;
			LeftOutState:=-100;
			LeftOut_MC_Stop.Execute:=FALSE;
			A_StopMC();
		ELSE
			LeftOutState:=1;
		END_IF
	1:
		LeftOut_MC_Stop.Execute:=TRUE;
		fb_ton_debug_7.IN:=TRUE;
		LeftOutState:=2;
	2:
		IF  NOT LeftOut_MC_Stop.Done THEN
				LeftOutState:=2;
		ELSE
			LeftOutState:=88;
			LeftOut_MC_Stop.Execute:=FALSE;
			A_StopMC();
		END_IF

	88:
		LeftOutStop:=FALSE;
		LeftOutState:=0;
		LeftOutBusy:=FALSE;
		LeftOutDone:=TRUE;
		Error:=FALSE;
		ErrorID:=0;
		fb_ton_debug_7.IN:=FALSE;

	-100:
		FB_PlcEmergencyStop();
		LeftOutStop:=FALSE;
		LeftOutState:=-100;
		LeftOutBusy:=FALSE;
		LeftOutDone:=FALSE;
		Error:=TRUE;
		LeftOut_MC_Stop.Execute:=FALSE;
		A_StopMC();
		fb_ton_debug_7.IN:=FALSE;

END_CASE
END_IF
END_ACTION

ACTION A_LeftTopStop:
IF LeftTopStop THEN
LeftTopBusy:=TRUE;
LeftTopDone:=FALSE;
fb_ton_debug_1(PT:=t#100ms);
A_StopMC();
CASE LeftTopState OF
	0:
		IF LeftTop_MC_Stop.Error THEN
			ErrorID:=41;
			LeftTopState:=-100;
			LeftTop_MC_Stop.Execute:=FALSE;
			A_StopMC();
		ELSE
			LeftTopState:=1;
		END_IF
	1:
		LeftTop_MC_Stop.Execute:=TRUE;
		fb_ton_debug_1.IN:=TRUE;
		LeftTopState:=2;
	2:
		IF  NOT LeftTop_MC_Stop.Done THEN
				LeftTopState:=2;
		ELSE
			LeftTopState:=88;
			LeftTop_MC_Stop.Execute:=FALSE;
			A_StopMC();
		END_IF

	88:
		LeftTopStop:=FALSE;
		LeftTopState:=0;
		LeftTopBusy:=FALSE;
		LeftTopDone:=TRUE;
		Error:=FALSE;
		ErrorID:=0;
		fb_ton_debug_1.IN:=FALSE;

	-100:
		FB_PlcEmergencyStop();
		LeftTopStop:=FALSE;
		LeftTopState:=-100;
		LeftTopBusy:=FALSE;
		LeftTopDone:=FALSE;
		Error:=TRUE;
		LeftTop_MC_Stop.Execute:=FALSE;
		A_StopMC();
		fb_ton_debug_1.IN:=FALSE;

END_CASE
END_IF
END_ACTION

ACTION A_OutStop:
IF OutStop THEN
OutBusy:=TRUE;
OutDone:=FALSE;
fb_ton4(PT:=T#100MS);
A_StopMC();
CASE OutState OF
	0:
		IF LeftOut_MC_Stop.Error OR RightOutLin_MC_Stop.Error THEN
			ErrorID:=1;
			OutState:=-100;
			LeftOut_MC_Stop.Execute:=FALSE;
			RightOutLin_MC_Stop.Execute:=FALSE;
			A_StopMC();
		ELSE
			OutState:=1;
		END_IF
	1:
		LeftOut_MC_Stop.Execute:=TRUE;
		RightOutLin_MC_Stop.Execute:=TRUE;
		fb_ton4.IN:=TRUE;
		OutState:=2;
	2:
		IF  NOT LeftOut_MC_Stop.Done OR NOT LeftOut_MC_Stop.Done THEN
				OutState:=2;
		ELSE
			OutState:=88;
			LeftOut_MC_Stop.Execute:=FALSE;
			RightOutLin_MC_Stop.Execute:=FALSE;
			A_StopMC();
		END_IF

	88:
		OutStop:=FALSE;
		OutState:=0;
		OutBusy:=FALSE;
		OutDone:=TRUE;
		Error:=FALSE;
		ErrorID:=0;
		fb_ton4.IN:=FALSE;

	-100:
		FB_PlcEmergencyStop();
		OutStop:=FALSE;
		OutState:=-100;
		OutBusy:=FALSE;
		OutDone:=FALSE;
		Error:=TRUE;
		LeftOut_MC_Stop.Execute:=FALSE;
		RightOutLin_MC_Stop.Execute:=FALSE;
		A_StopMC();
		fb_ton4.IN:=FALSE;

END_CASE
END_IF
END_ACTION

ACTION A_RightBottomStop:
IF RightBottomStop THEN
RightBottomBusy:=TRUE;
RightBottomDone:=FALSE;
fb_ton_debug_4(PT:=t#100ms);
A_StopMC();
CASE RightBottomState OF
	0:
		IF RightBottomLin_MC_Stop.Error THEN
			ErrorID:=41;
			RightBottomState:=-100;
			RightBottomLin_MC_Stop.Execute:=FALSE;
			A_StopMC();
		ELSE
			RightBottomState:=1;
		END_IF
	1:
		RightBottomLin_MC_Stop.Execute:=TRUE;
		fb_ton_debug_4.IN:=TRUE;
		RightBottomState:=2;
	2:
		IF  NOT RightBottomLin_MC_Stop.Done THEN
				RightBottomState:=2;
		ELSE
			RightBottomState:=88;
			RightBottomLin_MC_Stop.Execute:=FALSE;
			A_StopMC();
		END_IF

	88:
		RightBottomStop:=FALSE;
		RightBottomState:=0;
		RightBottomBusy:=FALSE;
		RightBottomDone:=TRUE;
		Error:=FALSE;
		ErrorID:=0;
		fb_ton_debug_4.IN:=FALSE;

	-100:
		FB_PlcEmergencyStop();
		RightBottomStop:=FALSE;
		RightBottomState:=-100;
		RightBottomBusy:=FALSE;
		RightBottomDone:=FALSE;
		Error:=TRUE;
		RightBottomLin_MC_Stop.Execute:=FALSE;
		A_StopMC();
		fb_ton_debug_4.IN:=FALSE;

END_CASE
END_IF
END_ACTION

ACTION A_RightInStop:
IF RightInStop THEN
RightInBusy:=TRUE;
RightInDone:=FALSE;
fb_ton_debug_6(PT:=t#100ms);
A_StopMC();
CASE RightInState OF
	0:
		IF RightInLin_MC_Stop.Error THEN
			ErrorID:=41;
			RightInState:=-100;
			RightInLin_MC_Stop.Execute:=FALSE;
			A_StopMC();
		ELSE
			RightInState:=1;
		END_IF
	1:
		RightInLin_MC_Stop.Execute:=TRUE;
		fb_ton_debug_6.IN:=TRUE;
		RightInState:=2;
	2:
		IF  NOT RightInLin_MC_Stop.Done THEN
				RightInState:=2;
		ELSE
			RightInState:=88;
			RightInLin_MC_Stop.Execute:=FALSE;
			A_StopMC();
		END_IF

	88:
		RightInStop:=FALSE;
		RightInState:=0;
		RightInBusy:=FALSE;
		RightInDone:=TRUE;
		Error:=FALSE;
		ErrorID:=0;
		fb_ton_debug_6.IN:=FALSE;

	-100:
		FB_PlcEmergencyStop();
		RightInStop:=FALSE;
		RightInState:=-100;
		RightInBusy:=FALSE;
		RightInDone:=FALSE;
		Error:=TRUE;
		RightInLin_MC_Stop.Execute:=FALSE;
		A_StopMC();
		fb_ton_debug_6.IN:=FALSE;

END_CASE
END_IF
END_ACTION

ACTION A_RightOutStop:
IF RightOutStop THEN
RightOutBusy:=TRUE;
RightOutDone:=FALSE;
fb_ton_debug_8(PT:=t#100ms);
A_StopMC();
CASE RightOutState OF
	0:
		IF RightOutLin_MC_Stop.Error THEN
			ErrorID:=41;
			RightOutState:=-100;
			RightOutLin_MC_Stop.Execute:=FALSE;
			A_StopMC();
		ELSE
			RightOutState:=1;
		END_IF
	1:
		RightOutLin_MC_Stop.Execute:=TRUE;
		fb_ton_debug_8.IN:=TRUE;
		RightOutState:=2;
	2:
		IF  NOT RightOutLin_MC_Stop.Done THEN
				RightOutState:=2;
		ELSE
			RightOutState:=88;
			RightOutLin_MC_Stop.Execute:=FALSE;
			A_StopMC();
		END_IF

	88:
		RightOutStop:=FALSE;
		RightOutState:=0;
		RightOutBusy:=FALSE;
		RightOutDone:=TRUE;
		Error:=FALSE;
		ErrorID:=0;
		fb_ton_debug_8.IN:=FALSE;

	-100:
		FB_PlcEmergencyStop();
		RightOutStop:=FALSE;
		RightOutState:=-100;
		RightOutBusy:=FALSE;
		RightOutDone:=FALSE;
		Error:=TRUE;
		RightOutLin_MC_Stop.Execute:=FALSE;
		A_StopMC();
		fb_ton_debug_8.IN:=FALSE;

END_CASE
END_IF
END_ACTION

ACTION A_RightTopStop:
IF RightTopStop THEN
RightTopBusy:=TRUE;
RightTopDone:=FALSE;
fb_ton_debug_2(PT:=t#100ms);
A_StopMC();
CASE RightTopState OF
	0:
		IF RightTopLin_MC_Stop.Error THEN
			ErrorID:=41;
			RightTopState:=-100;
			RightTopLin_MC_Stop.Execute:=FALSE;
			A_StopMC();
		ELSE
			RightTopState:=1;
		END_IF
	1:
		RightTopLin_MC_Stop.Execute:=TRUE;
		fb_ton_debug_2.IN:=TRUE;
		RightTopState:=2;
	2:
		IF  NOT RightTopLin_MC_Stop.Done THEN
				RightTopState:=2;
		ELSE
			RightTopState:=88;
			RightTopLin_MC_Stop.Execute:=FALSE;
			A_StopMC();
		END_IF

	88:
		RightTopStop:=FALSE;
		RightTopState:=0;
		RightTopBusy:=FALSE;
		RightTopDone:=TRUE;
		Error:=FALSE;
		ErrorID:=0;
		fb_ton_debug_2.IN:=FALSE;

	-100:
		FB_PlcEmergencyStop();
		RightTopStop:=FALSE;
		RightTopState:=-100;
		RightTopBusy:=FALSE;
		RightTopDone:=FALSE;
		Error:=TRUE;
		RightTopLin_MC_Stop.Execute:=FALSE;
		A_StopMC();
		fb_ton_debug_2.IN:=FALSE;

END_CASE
END_IF
END_ACTION

ACTION A_StopMC:
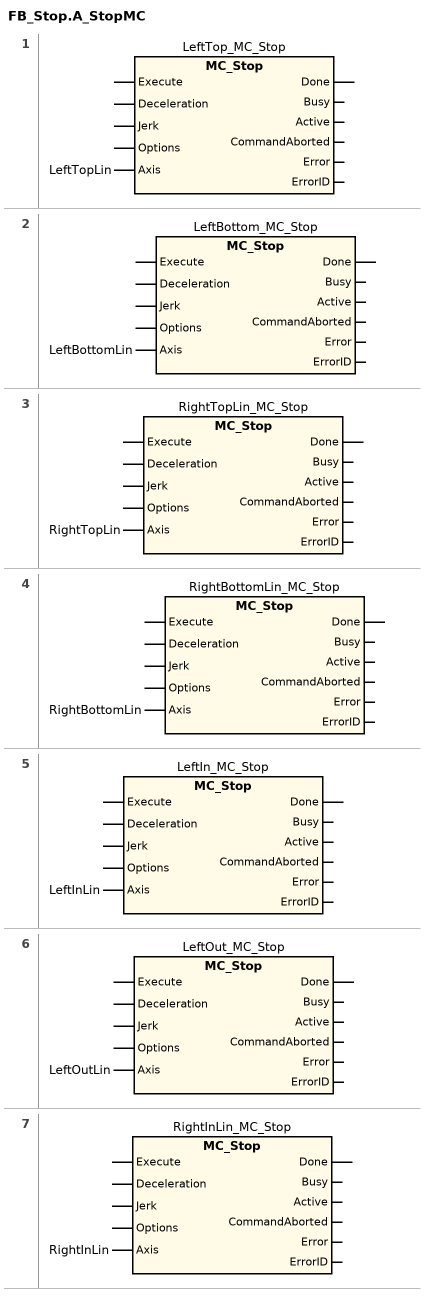
// NETWORK 1
LeftTop_MC_Stop(Axis := LeftTopLin); // MC_Stop

// NETWORK 2
LeftBottom_MC_Stop(Axis := LeftBottomLin); // MC_Stop

// NETWORK 3
RightTopLin_MC_Stop(Axis := RightTopLin); // MC_Stop

// NETWORK 4
RightBottomLin_MC_Stop(Axis := RightBottomLin); // MC_Stop

// NETWORK 5
LeftIn_MC_Stop(Axis := LeftInLin); // MC_Stop

// NETWORK 6
LeftOut_MC_Stop(Axis := LeftOutLin); // MC_Stop

// NETWORK 7
RightInLin_MC_Stop(Axis := RightInLin); // MC_Stop

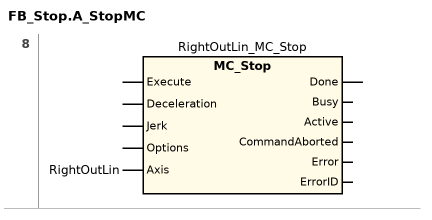
// NETWORK 8
RightOutLin_MC_Stop(Axis := RightOutLin); // MC_Stop
END_ACTION

ACTION A_TopStop:
IF TopStop THEN
TopBusy:=TRUE;
TopDone:=FALSE;
fb_ton1(PT:=t#100ms);
A_StopMC();
CASE TopState OF
	0:
		IF LeftTop_MC_Stop.Error OR RightTopLin_MC_Stop.Error THEN
			ErrorID:=1;
			TopState:=-100;
			LeftTop_MC_Stop.Execute:=FALSE;
			A_StopMC();
		ELSE
			TopState:=1;
		END_IF
	1:
		LeftTop_MC_Stop.Execute:=TRUE;
		RightTopLin_MC_Stop.Execute:=TRUE;
		fb_ton1.IN:=TRUE;
		TopState:=2;
	2:
		IF  NOT LeftTop_MC_Stop.Done OR NOT RightTopLin_MC_Stop.Done THEN
				TopState:=2;
		ELSE
			TopState:=88;
			LeftTop_MC_Stop.Execute:=FALSE;
			RightTopLin_MC_Stop.Execute:=FALSE;
			A_StopMC();
		END_IF

	88:
		TopStop:=FALSE;
		TopState:=0;
		TopBusy:=FALSE;
		TopDone:=TRUE;
		Error:=FALSE;
		ErrorID:=0;
		fb_ton1.IN:=FALSE;

	-100:
		FB_PlcEmergencyStop();
		TopStop:=FALSE;
		TopState:=-100;
		TopBusy:=FALSE;
		TopDone:=FALSE;
		Error:=TRUE;
		LeftTop_MC_Stop.Execute:=FALSE;
		RightTopLin_MC_Stop.Execute:=FALSE;
		A_StopMC();
		fb_ton1.IN:=FALSE;

END_CASE
END_IF
END_ACTION

END_FUNCTION_BLOCK

// ---- POUs/2.SingleMotorMode/DebugMode/DebugMode.TcPOU
PROGRAM DebugMode
VAR
(* Common*)
	d_state: DINT;(*PowerOffState*)
	InitDone:BOOL;
	Busy: BOOL;
	fb_ton: TON;
	PowerState: INT;(*PowerOnState*)
	ton_t: TON;
(*Key Command*)
	LeftTopLinPositionNew:LREAL:=10;
	LeftTopLinVelocityNew:LREAL:=0.2;
	btn_LeftTopLinMove:BOOL;
	btn_LeftTopLinStop:BOOL;
	RightTopLinPositionNew:LREAL:=10;
	RightTopLinVelocityNew:LREAL:=0.2;
	btn_RightTopLinMove:BOOL;
	btn_RightTopLinStop:BOOL;
	LeftBottomLinPositionNew:LREAL:=10;
	LeftBottomLinVelocityNew:LREAL:=0.2;
	btn_LeftBottomLinMove:BOOL;
	btn_LeftBottomLinStop:BOOL;
	RightBottomLinPositionNew:LREAL:=10;
	RightBottomLinVelocityNew:LREAL:=0.2;
	btn_RightBottomLinMove:BOOL;
	btn_RightBottomLinStop:BOOL;
	
	
	LeftInLinPositionNew:LREAL:=10;
	LeftInLinVelocityNew:LREAL:=0.2;
	btn_LeftInLinMove:BOOL;
	btn_LeftInLinStop:BOOL;
	RightInLinPositionNew:LREAL:=10;
	RightInLinVelocityNew:LREAL:=0.2;
	btn_RightInLinMove:BOOL;
	btn_RightInLinStop:BOOL;
	LeftOutLinPositionNew:LREAL:=10;
	LeftOutLinVelocityNew:LREAL:=0.2;
	btn_LeftOutLinMove:BOOL;
	btn_LeftOutLinStop:BOOL;
	RightOutLinPositionNew:LREAL:=10;
	RightOutLinVelocityNew:LREAL:=0.2;
	btn_RightOutLinMove:BOOL;
	btn_RightOutLinStop:BOOL;
(*LeftTopLin*)
	fb_ton1_1:TON;
	fb_ton1_2:TON;
	LeftTopLinState:DINT;
	LeftTopLinBusy:BOOL;
	LeftTopLin_m_state: DINT;
	LeftTopLin_s_state: DINT;
(*RightTopLin*)
	fb_ton2_1:TON;
	fb_ton2_2:TON;
	RightTopLinState:DINT;
	RightTopLinBusy:BOOL;
	RightTopLin_m_state: DINT;
	RightTopLin_s_state: DINT;
(*LeftBottomLin*)
	fb_ton3_1:TON;
	fb_ton3_2:TON;
	LeftBottomLinState:DINT;
	LeftBottomLinBusy:BOOL;
	LeftBottomLin_m_state: DINT;
	LeftBottomLin_s_state: DINT;
(*RightBottomLin*)
	fb_ton4_1:TON;
	fb_ton4_2:TON;
	RightBottomLinState:DINT;
	RightBottomLinBusy:BOOL;
	RightBottomLin_m_state: DINT;
	RightBottomLin_s_state: DINT;
	
(*LeftInLin*)
	fb_ton5_1:TON;
	fb_ton5_2:TON;
	LeftInLinState:DINT;
	LeftInLinBusy:BOOL;
	LeftInLin_m_state: DINT;
	LeftInLin_s_state: DINT;
(*RightInLin*)
	fb_ton6_1:TON;
	fb_ton6_2:TON;
	RightInLinState:DINT;
	RightInLinBusy:BOOL;
	RightInLin_m_state: DINT;
	RightInLin_s_state: DINT;
(*LeftOutLin*)
	fb_ton7_1:TON;
	fb_ton7_2:TON;
	LeftOutLinState:DINT;
	LeftOutLinBusy:BOOL;
	LeftOutLin_m_state: DINT;
	LeftOutLin_s_state: DINT;
(*RightOutLin*)
	fb_ton8_1:TON;
	fb_ton8_2:TON;
	RightOutLinState:DINT;
	RightOutLinBusy:BOOL;
	RightOutLin_m_state: DINT;
	RightOutLin_s_state: DINT;


	btn_LeftTopStop: BOOL;
	(*¼ì²âµ½ÏÞÎ»£¬»Ö¸´Move×´Ì¬*)
	FTrig_ReachLS: F_TRIG;
	FTrig_btn_GapMove: F_TRIG;
END_VAR

(*********Monitor All Carrirt Position**********************)
A_MonitoringAllAxis();
(*********A_PosDiffDetection********************************)
A_PosDiffDetection();
(*********btn_PowerOn***************************************)
IF st_Power=1 THEN
	InitDone:=TRUE;
END_IF
IF btn_Power AND st_Power=0 THEN
	btn_PowerOn:=TRUE;
	btn_Power:=FALSE;
END_IF
IF btn_Power AND st_Power=1 THEN
	btn_PowerOff:=TRUE;
	btn_Power:=FALSE;
END_IF
(**********btn_PowerOn****************************************)
IF btn_PowerOn THEN
	A_PowerOn();
END_IF
IF btn_PowerOff THEN
	A_PowerOff();
END_IF

(**************btn_PowerOff*******************************)
IF btn_PowerOff THEN
	A_PowerOff();
END_IF

(**********************MOVE****************)
A_DebugMove();
(**********************STOP***************)
A_DebugStop();

FTrig_ReachLS(CLK:=Unreach_LS_Far AND Unreach_LS_Near);
IF FTrig_ReachLS.Q THEN
	btn_LeftTopLinStop:=TRUE;
	btn_RightTopLinStop:=TRUE;
	btn_LeftBottomLinStop:=TRUE;
	btn_RightBottomLinStop:=TRUE;
	btn_LeftInLinStop:=TRUE;
	btn_RightInLinStop:=TRUE;
	btn_LeftOutLinStop:=TRUE;
	btn_RightOutLinStop:=TRUE;
END_IF

ACTION A_DebugMove:
(*********************************************************************LeftTop_MOVE*****************************************************************)
IF InitDone THEN
	IF btn_LeftTopLinMove THEN
		CASE LeftTopLin_m_state OF
			0:
				FB_Move.Mode:=2;
				FB_Move.CoupleState:=st_Couple;	
				FB_Move.PowerState:=st_Power;	
				FB_Move.LeftTopMove:=TRUE;	
				FB_Move.LeftTopPosition:=LeftTopLinPositionNew;
				FB_Move.LeftTopVelocity:=LeftTopLinVelocityNew;	
				FB_Move();								
				LeftTopLin_m_state:=1;
			1:
				FB_Move();
				IF NOT FB_Move.LeftTopDone THEN
					LeftTopLin_m_state:=1;
					LED_Run:=TRUE;
				ELSE									
					LeftTopLin_m_state:=88;
				END_IF

			88:
				btn_LeftTopLinMove:=FALSE;
				LeftTopLin_m_state:=0;
				LED_Run:=FALSE;
		END_CASE
	END_IF
END_IF

(*********************************************************************RightTop_MOVE*****************************************************************)
IF InitDone THEN
	IF btn_RightTopLinMove THEN
		CASE RightTopLin_m_state OF
			0:
				FB_Move.Mode:=2;	
				FB_Move.CoupleState:=st_Couple;	
				FB_Move.PowerState:=st_Power;	
				FB_Move.RightTopMove:=TRUE;	
				FB_Move.RightTopPosition:=RightTopLinPositionNew;
				FB_Move.RightTopVelocity:=RightTopLinVelocityNew;
				FB_Move();
				RightTopLin_m_state:=1;
			1:
				FB_Move();
				IF NOT FB_Move.RightTopDone THEN
					RightTopLin_m_state:=1;
					LED_Run:=TRUE;
				ELSE
					RightTopLin_m_state:=88;
				END_IF

			88:
				btn_RightTopLinMove:=FALSE;	
				RightTopLin_m_state:=0;
				LED_Run:=FALSE;
		END_CASE
	END_IF
END_IF

(*********************************************************************LeftBottom_MOVE*****************************************************************)
IF InitDone THEN
	IF btn_LeftBottomLinMove THEN
		CASE LeftBottomLin_m_state OF
			0:
				FB_Move.Mode:=2;	
				FB_Move.CoupleState:=st_Couple;	
				FB_Move.PowerState:=st_Power;
				FB_Move.LeftBottomMove:=TRUE;
				FB_Move.LeftBottomPosition:=LeftBottomLinPositionNew;
				FB_Move.LeftBottomVelocity:=LeftBottomLinVelocityNew;
				FB_Move();	
				LeftBottomLin_m_state:=1;
			1:
				FB_Move();
				IF NOT FB_Move.LeftBottomDone THEN	
					LeftBottomLin_m_state:=1;
					LED_Run:=TRUE;
				ELSE
					LeftBottomLin_m_state:=88;
				END_IF

			88:
				btn_LeftBottomLinMove:=FALSE;
				LeftBottomLin_m_state:=0;
				LED_Run:=FALSE;
		END_CASE
	END_IF
END_IF

(*********************************************************************RightBottom_MOVE*****************************************************************)
IF InitDone THEN
	IF btn_RightBottomLinMove THEN
		CASE RightBottomLin_m_state OF
			0:
				FB_Move.Mode:=2;
				FB_Move.CoupleState:=st_Couple;	
				FB_Move.PowerState:=st_Power;
				FB_Move.RightBottomMove:=TRUE;
				FB_Move.RightBottomPosition:=RightBottomLinPositionNew;
				FB_Move.RightBottomVelocity:=RightBottomLinVelocityNew;	
				FB_Move();	
				RightBottomLin_m_state:=1;
			1:
				FB_Move();
				IF NOT FB_Move.RightBottomDone THEN	
					RightBottomLin_m_state:=1;
					LED_Run:=TRUE;
				ELSE	
					RightBottomLin_m_state:=88;
				END_IF

			88:
				btn_RightBottomLinMove:=FALSE;
				RightBottomLin_m_state:=0;
				LED_Run:=FALSE;
		END_CASE
	END_IF
END_IF

(*********************************************************************LeftIn_MOVE*****************************************************************)
IF InitDone THEN
	IF btn_LeftInLinMove THEN
		CASE LeftInLin_m_state OF
			0:
				FB_Move.Mode:=2;
				FB_Move.CoupleState:=st_Couple;	
				FB_Move.PowerState:=st_Power;	
				FB_Move.LeftInMove:=TRUE;	
				FB_Move.LeftInPosition:=LeftInLinPositionNew;
				FB_Move.LeftInVelocity:=LeftInLinVelocityNew;	
				FB_Move();								
				LeftInLin_m_state:=1;
			1:
				FB_Move();
				IF NOT FB_Move.LeftInDone THEN
					LeftInLin_m_state:=1;
					LED_Run:=TRUE;
				ELSE									
					LeftInLin_m_state:=88;
				END_IF

			88:
				btn_LeftInLinMove:=FALSE;
				LeftInLin_m_state:=0;
				LED_Run:=FALSE;
		END_CASE
	END_IF
END_IF

(*********************************************************************RightIn_MOVE*****************************************************************)
IF InitDone THEN
	IF btn_RightInLinMove THEN
		CASE RightInLin_m_state OF
			0:
				FB_Move.Mode:=2;	
				FB_Move.CoupleState:=st_Couple;	
				FB_Move.PowerState:=st_Power;	
				FB_Move.RightInMove:=TRUE;	
				FB_Move.RightInPosition:=RightInLinPositionNew;
				FB_Move.RightInVelocity:=RightInLinVelocityNew;
				FB_Move();
				RightInLin_m_state:=1;
			1:
				FB_Move();
				IF NOT FB_Move.RightInDone THEN
					RightInLin_m_state:=1;
					LED_Run:=TRUE;
				ELSE
					RightInLin_m_state:=88;
				END_IF

			88:
				btn_RightInLinMove:=FALSE;	
				RightInLin_m_state:=0;
				LED_Run:=FALSE;
		END_CASE
	END_IF
END_IF

(*********************************************************************LeftOut_MOVE*****************************************************************)
IF InitDone THEN
	IF btn_LeftOutLinMove THEN
		CASE LeftOutLin_m_state OF
			0:
				FB_Move.Mode:=2;	
				FB_Move.CoupleState:=st_Couple;	
				FB_Move.PowerState:=st_Power;
				FB_Move.LeftOutMove:=TRUE;
				FB_Move.LeftOutPosition:=LeftOutLinPositionNew;
				FB_Move.LeftOutVelocity:=LeftOutLinVelocityNew;
				FB_Move();	
				LeftOutLin_m_state:=1;
			1:
				FB_Move();
				IF NOT FB_Move.LeftOutDone THEN	
					LeftOutLin_m_state:=1;
					LED_Run:=TRUE;
				ELSE
					LeftOutLin_m_state:=88;
				END_IF

			88:
				btn_LeftOutLinMove:=FALSE;
				LeftOutLin_m_state:=0;
				LED_Run:=FALSE;
		END_CASE
	END_IF
END_IF

(*********************************************************************RightOut_MOVE*****************************************************************)
IF InitDone THEN
	IF btn_RightOutLinMove THEN
		CASE RightOutLin_m_state OF
			0:
				FB_Move.Mode:=2;
				FB_Move.CoupleState:=st_Couple;	
				FB_Move.PowerState:=st_Power;
				FB_Move.RightOutMove:=TRUE;
				FB_Move.RightOutPosition:=RightOutLinPositionNew;
				FB_Move.RightOutVelocity:=RightOutLinVelocityNew;	
				FB_Move();	
				RightOutLin_m_state:=1;
			1:
				FB_Move();
				IF NOT FB_Move.RightOutDone THEN	
					RightOutLin_m_state:=1;
					LED_Run:=TRUE;
				ELSE	
					RightOutLin_m_state:=88;
				END_IF

			88:
				btn_RightOutLinMove:=FALSE;
				RightOutLin_m_state:=0;
				LED_Run:=FALSE;
		END_CASE
	END_IF
END_IF
END_ACTION

ACTION A_DebugStop:
(*******************************************************************LeftTop_STOP********************************************************************)
IF btn_LeftTopLinStop THEN
	LED_Run:=FALSE;
	FB_Move.LeftTopReset:=TRUE;	
	FB_Move();	
	btn_LeftTopLinMove:=FALSE;	
	LeftTopLin_m_state:=0;	
	CASE LeftTopLin_s_state OF
			0:
				FB_Stop.Mode:=2;
				FB_Stop.CoupleState:=st_Couple;	
				FB_Stop.PowerState:=st_Power;	
				FB_Stop.LeftTopStop:=TRUE;
				FB_Stop();	
				LeftTopLin_s_state:=1;
			1:
				FB_Stop();
				IF NOT FB_Stop.LeftTopDone THEN	
					LeftTopLin_s_state:=1;
				ELSE
					LeftTopLin_s_state:=88;
				END_IF
			88:
				btn_LeftTopLinStop:=FALSE;	
				FB_Move.LeftTopReset:=FALSE;	
				LeftTopLin_s_state:=0;
		END_CASE

END_IF

(*******************************************************************RightTop_STOP********************************************************************)
IF btn_RightTopLinStop THEN
	LED_Run:=FALSE;
	FB_Move.RightTopReset:=TRUE;
	FB_Move();
	btn_RightTopLinMove:=FALSE;	
	RightTopLin_m_state:=0;		
	CASE RightTopLin_s_state OF
			0:
				FB_Stop.Mode:=2;
				FB_Stop.CoupleState:=st_Couple;
				FB_Stop.PowerState:=st_Power;
				FB_Stop.RightTopStop:=TRUE;
				FB_Stop();
				RightTopLin_s_state:=1;
			1:
				FB_Stop();
				IF NOT FB_Stop.RightTopDone THEN
					RightTopLin_s_state:=1;
				ELSE	
					RightTopLin_s_state:=88;
				END_IF
			88:
				btn_RightTopLinStop:=FALSE;	
				FB_Move.RightTopReset:=FALSE;
				RightTopLin_s_state:=0;
		END_CASE

END_IF

(*******************************************************************LeftBottom_STOP********************************************************************)
IF btn_LeftBottomLinStop THEN
	LED_Run:=FALSE;
	FB_Move.LeftBottomReset:=TRUE;
	FB_Move();						
	btn_LeftBottomLinMove:=FALSE;		
	LeftBottomLin_m_state:=0;		
	CASE LeftBottomLin_s_state OF
			0:
				FB_Stop.Mode:=2;
				FB_Stop.CoupleState:=st_Couple;
				FB_Stop.PowerState:=st_Power;
				FB_Stop.LeftBottomStop:=TRUE;	
				FB_Stop();	
				LeftBottomLin_s_state:=1;
			1:
				FB_Stop();
				IF NOT FB_Stop.LeftBottomDone THEN
					LeftBottomLin_s_state:=1;
				ELSE
					LeftBottomLin_s_state:=88;
				END_IF
			88:
				btn_LeftBottomLinStop:=FALSE;
				FB_Move.LeftBottomReset:=FALSE;	
				LeftBottomLin_s_state:=0;
		END_CASE

END_IF

(*******************************************************************RightBottom_STOP********************************************************************)
IF btn_RightBottomLinStop THEN
	LED_Run:=FALSE;
	FB_Move.RightBottomReset:=TRUE;
	FB_Move();	
	btn_RightBottomLinMove:=FALSE;
	RightBottomLin_m_state:=0;	
	CASE RightBottomLin_s_state OF
			0:
				FB_Stop.Mode:=2;
				FB_Stop.CoupleState:=st_Couple;	
				FB_Stop.PowerState:=st_Power;
				FB_Stop.RightBottomStop:=TRUE;	
				FB_Stop();
				RightBottomLin_s_state:=1;
			1:
				FB_Stop();
				IF NOT FB_Stop.RightBottomDone THEN
					RightBottomLin_s_state:=1;
				ELSE
					RightBottomLin_s_state:=88;
				END_IF
			88:
				btn_RightBottomLinStop:=FALSE;
				FB_Move.RightBottomReset:=FALSE;
				RightBottomLin_s_state:=0;
		END_CASE

END_IF

(*******************************************************************LeftIn_STOP********************************************************************)
IF btn_LeftInLinStop THEN
	LED_Run:=FALSE;
	FB_Move.LeftInReset:=TRUE;	
	FB_Move();	
	btn_LeftInLinMove:=FALSE;	
	LeftInLin_m_state:=0;	
	CASE LeftInLin_s_state OF
			0:
				FB_Stop.Mode:=2;
				FB_Stop.CoupleState:=st_Couple;	
				FB_Stop.PowerState:=st_Power;	
				FB_Stop.LeftInStop:=TRUE;
				FB_Stop();	
				LeftInLin_s_state:=1;
			1:
				FB_Stop();
				IF NOT FB_Stop.LeftInDone THEN	
					LeftInLin_s_state:=1;
				ELSE
					LeftInLin_s_state:=88;
				END_IF
			88:
				btn_LeftInLinStop:=FALSE;	
				FB_Move.LeftInReset:=FALSE;	
				LeftInLin_s_state:=0;
		END_CASE

END_IF

(*******************************************************************RightIn_STOP********************************************************************)
IF btn_RightInLinStop THEN
	LED_Run:=FALSE;
	FB_Move.RightInReset:=TRUE;
	FB_Move();
	btn_RightInLinMove:=FALSE;	
	RightInLin_m_state:=0;		
	CASE RightInLin_s_state OF
			0:
				FB_Stop.Mode:=2;
				FB_Stop.CoupleState:=st_Couple;
				FB_Stop.PowerState:=st_Power;
				FB_Stop.RightInStop:=TRUE;
				FB_Stop();
				RightInLin_s_state:=1;
			1:
				FB_Stop();
				IF NOT FB_Stop.RightInDone THEN
					RightInLin_s_state:=1;
				ELSE	
					RightInLin_s_state:=88;
				END_IF
			88:
				btn_RightInLinStop:=FALSE;	
				FB_Move.RightInReset:=FALSE;
				RightInLin_s_state:=0;
		END_CASE

END_IF

(*******************************************************************LeftOut_STOP********************************************************************)
IF btn_LeftOutLinStop THEN
	LED_Run:=FALSE;
	FB_Move.LeftOutReset:=TRUE;
	FB_Move();						
	btn_LeftOutLinMove:=FALSE;		
	LeftOutLin_m_state:=0;		
	CASE LeftOutLin_s_state OF
			0:
				FB_Stop.Mode:=2;
				FB_Stop.CoupleState:=st_Couple;
				FB_Stop.PowerState:=st_Power;
				FB_Stop.LeftOutStop:=TRUE;	
				FB_Stop();	
				LeftOutLin_s_state:=1;
			1:
				FB_Stop();
				IF NOT FB_Stop.LeftOutDone THEN
					LeftOutLin_s_state:=1;
				ELSE
					LeftOutLin_s_state:=88;
				END_IF
			88:
				btn_LeftOutLinStop:=FALSE;
				FB_Move.LeftOutReset:=FALSE;	
				LeftOutLin_s_state:=0;
		END_CASE

END_IF

(*******************************************************************RightOut_STOP********************************************************************)
IF btn_RightOutLinStop THEN
	LED_Run:=FALSE;
	FB_Move.RightOutReset:=TRUE;
	FB_Move();	
	btn_RightOutLinMove:=FALSE;
	RightOutLin_m_state:=0;	
	CASE RightOutLin_s_state OF
			0:
				FB_Stop.Mode:=2;
				FB_Stop.CoupleState:=st_Couple;	
				FB_Stop.PowerState:=st_Power;
				FB_Stop.RightOutStop:=TRUE;	
				FB_Stop();
				RightOutLin_s_state:=1;
			1:
				FB_Stop();
				IF NOT FB_Stop.RightOutDone THEN
					RightOutLin_s_state:=1;
				ELSE
					RightOutLin_s_state:=88;
				END_IF
			88:
				btn_RightOutLinStop:=FALSE;
				FB_Move.RightOutReset:=FALSE;
				RightOutLin_s_state:=0;
		END_CASE

END_IF
END_ACTION

ACTION A_monitoringAllAxis:
(*************************************************************************************2.4Öá¹âÕ¤³ßÎ»ÖÃ¡¢ËÙ¶È¶Ô±È¼ì²é**********************************************************************)
IF st_power<>0 THEN

IF ABS(Pos_LeftTopLin-Pos_LeftBottomLin)>Threshold_TBLeftPos_Debug  THEN
		btn_LeftTopLinStop:=TRUE;
		btn_RightTopLinStop:=TRUE;
		btn_LeftBottomLinStop:=TRUE;
		btn_RightBottomLInStop:=TRUE;
		FB_PlcEmergencyStop();
		Error:=TRUE;
		ErrorID:=11;
		LED_Error:=TRUE;
END_IF

IF ABS(Pos_RightTopLin-Pos_RightBottomLin)>Threshold_TBRightPos_Debug  THEN
		btn_LeftTopLinStop:=TRUE;
		btn_RightTopLinStop:=TRUE;
		btn_LeftBottomLinStop:=TRUE;
		btn_RightBottomLInStop:=TRUE;
		FB_PlcEmergencyStop();
		Error:=TRUE;
		ErrorID:=12;
		LED_Error:=TRUE;
END_IF

IF ABS(Pos_LeftTopLin-Pos_RightTopLin)>Threshold_TopPos_Debug  THEN
		btn_LeftTopLinStop:=TRUE;
		btn_RightTopLinStop:=TRUE;
		btn_LeftBottomLinStop:=TRUE;
		btn_RightBottomLInStop:=TRUE;
		FB_PlcEmergencyStop();
		Error:=TRUE;
		ErrorID:=13;
		LED_Error:=TRUE;
END_IF

IF ABS(Pos_LeftBottomLin-Pos_RightBottomLin)>Threshold_BottomPos_Debug  THEN
		btn_LeftTopLinStop:=TRUE;
		btn_RightTopLinStop:=TRUE;
		btn_LeftBottomLinStop:=TRUE;
		btn_RightBottomLInStop:=TRUE;
		FB_PlcEmergencyStop();
		Error:=TRUE;
		ErrorID:=14;
		LED_Error:=TRUE;
END_IF
//

IF ABS(Pos_LeftInLin-Pos_LeftOutLin)>Threshold_IOLeftPos_Debug  THEN
		btn_LeftInLinStop:=TRUE;
		btn_RightInLinStop:=TRUE;
		btn_LeftOutLinStop:=TRUE;
		btn_RightOutLInStop:=TRUE;
		FB_PlcEmergencyStop();
		Error:=TRUE;
		ErrorID:=15;
		LED_Error:=TRUE;
END_IF

IF ABS(Pos_RightInLin-Pos_RightOutLin)>Threshold_IORightPos_Debug  THEN
		btn_LeftInLinStop:=TRUE;
		btn_RightInLinStop:=TRUE;
		btn_LeftOutLinStop:=TRUE;
		btn_RightOutLInStop:=TRUE;
		FB_PlcEmergencyStop();
		Error:=TRUE;
		ErrorID:=16;
		LED_Error:=TRUE;
END_IF

IF ABS(Pos_LeftInLin-Pos_RightInLin)>Threshold_InPos_Debug  THEN
		btn_LeftInLinStop:=TRUE;
		btn_RightInLinStop:=TRUE;
		btn_LeftOutLinStop:=TRUE;
		btn_RightOutLInStop:=TRUE;
		FB_PlcEmergencyStop();
		Error:=TRUE;
		ErrorID:=17;
		LED_Error:=TRUE;
END_IF

IF ABS(Pos_LeftOutLin-Pos_RightOutLin)>Threshold_OutPos_Debug  THEN
		btn_LeftInLinStop:=TRUE;
		btn_RightInLinStop:=TRUE;
		btn_LeftOutLinStop:=TRUE;
		btn_RightOutLInStop:=TRUE;
		FB_PlcEmergencyStop();
		Error:=TRUE;
		ErrorID:=18;
		LED_Error:=TRUE;
END_IF
END_IF
END_ACTION

ACTION A_PosDiffDetection:
IF ABS(PosDiff_LeftTopLin_actual-PosDiff_RightTopLin_actual)>0.2 THEN
	ErrorID:=51;
	Error:=TRUE;
	btn_LeftTopLinStop:=TRUE;
	btn_RightTopLinStop:=TRUE;
	btn_LeftBottomLinStop:=TRUE;
	btn_RightBottomLInStop:=TRUE;
	FB_PlcEmergencyStop();
	LED_Error:=TRUE;
ELSIF ABS(PosDiff_LeftBottomLin_actual-PosDiff_RightBottomLin_actual)>0.2 THEN
	ErrorID:=52;
	Error:=TRUE;
	btn_LeftTopLinStop:=TRUE;
	btn_RightTopLinStop:=TRUE;
	btn_LeftBottomLinStop:=TRUE;
	btn_RightBottomLInStop:=TRUE;
	FB_PlcEmergencyStop();
	LED_Error:=TRUE;
END_IF

IF ABS(PosDiff_LeftInLin_actual-PosDiff_RightInLin_actual)>0.2 THEN
	ErrorID:=53;
	Error:=TRUE;
	btn_LeftInLinStop:=TRUE;
	btn_RightInLinStop:=TRUE;
	btn_LeftOutLinStop:=TRUE;
	btn_RightOutLInStop:=TRUE;
	FB_PlcEmergencyStop();
	LED_Error:=TRUE;
ELSIF ABS(PosDiff_LeftOutLin_actual-PosDiff_RightOutLin_actual)>0.2 THEN
	ErrorID:=54;
	Error:=TRUE;
	btn_LeftInLinStop:=TRUE;
	btn_RightInLinStop:=TRUE;
	btn_LeftOutLinStop:=TRUE;
	btn_RightOutLInStop:=TRUE;
	FB_PlcEmergencyStop();
	LED_Error:=TRUE;
END_IF
END_ACTION

ACTION A_PowerOff:
CASE d_state OF
		0:(*PowerOff*)
			FB_Power(Off:=TRUE);
				d_state:=1;
		1:
			IF NOT FB_power.OffStatus THEN
				d_state:=1;
			ELSE
				d_state:=88;
			END_IF
		88:(*ResetAllState*)
			btn_PowerOn:=FALSE;
			btn_PowerOff:=FALSE;
			ton_t.IN:=FALSE;
			InitDone:=FALSE;
			Error:=FALSE;
			ErrorID:=0;
			d_state:=0;

			btn_LeftTopLinMove:=FALSE;
			btn_LeftTopLinStop:=FALSE;
			fb_ton1_1.IN:=FALSE;
			fb_ton1_2.IN:=FALSE;
			LeftTopLinState:=0;
			LeftTopLinBusy:=FALSE;
			LeftTopLin_m_state:=0;
			LeftTopLin_s_state:=0;

			btn_RightTopLinMove:=FALSE;
			btn_RightTopLinStop:=FALSE;
			fb_ton2_1.IN:=FALSE;
			fb_ton2_2.IN:=FALSE;
			RightTopLinState:=0;
			RightTopLinBusy:=FALSE;
			RightTopLin_m_state:=0;
			RightTopLin_s_state:=0;

			btn_LeftBottomLinMove:=FALSE;
			btn_LeftBottomLinStop:=FALSE;
			fb_ton3_1.IN:=FALSE;
			fb_ton3_2.IN:=FALSE;
			LeftBottomLinState:=0;
			LeftBottomLinBusy:=FALSE;
			LeftBottomLin_m_state:=0;
			LeftBottomLin_s_state:=0;

			btn_RightBottomLinMove:=FALSE;
			btn_RightBottomLinStop:=FALSE;
			fb_ton4_1.IN:=FALSE;
			fb_ton4_2.IN:=FALSE;
			RightBottomLinState:=0;
			RightBottomLinBusy:=FALSE;
			RightBottomLin_m_state:=0;
			RightBottomLin_s_state:=0;
			
			btn_LeftInLinMove:=FALSE;
			btn_LeftInLinStop:=FALSE;
			fb_ton5_1.IN:=FALSE;
			fb_ton5_2.IN:=FALSE;
			LeftInLinState:=0;
			LeftInLinBusy:=FALSE;
			LeftInLin_m_state:=0;
			LeftInLin_s_state:=0;

			btn_RightInLinMove:=FALSE;
			btn_RightInLinStop:=FALSE;
			fb_ton6_1.IN:=FALSE;
			fb_ton6_2.IN:=FALSE;
			RightInLinState:=0;
			RightInLinBusy:=FALSE;
			RightInLin_m_state:=0;
			RightInLin_s_state:=0;

			btn_LeftOutLinMove:=FALSE;
			btn_LeftOutLinStop:=FALSE;
			fb_ton7_1.IN:=FALSE;
			fb_ton7_2.IN:=FALSE;
			LeftBottomLinState:=0;
			LeftOutLinBusy:=FALSE;
			LeftOutLin_m_state:=0;
			LeftOutLin_s_state:=0;

			btn_RightOutLinMove:=FALSE;
			btn_RightOutLinStop:=FALSE;
			fb_ton8_1.IN:=FALSE;
			fb_ton8_2.IN:=FALSE;
			RightOutLinState:=0;
			RightOutLinBusy:=FALSE;
			RightOutLin_m_state:=0;
			RightOutLin_s_state:=0;

		LED_Error:=FALSE;
		LED_Run:=FALSE;

END_CASE
END_ACTION

ACTION A_PowerOn:
fb_ton(PT:=T#0.5S);
CASE PowerState OF
	0:	(*FB_Power_On*)
		FB_Power(On:=TRUE);
		fb_ton.IN:=TRUE;
		PowerState:=1;
	1:	(*wait*)
		FB_power();
		IF NOT FB_power.OnStatus THEN		(*FB_Power_OnÃ»ÓÐÖ´ÐÐÍê£¬wait£¬³¬Ê±FB Error*)
			IF NOT fb_ton.Q THEN
				PowerState:=1;
			ELSE
				ErrorID:=1;
				PowerState:=99;
			END_IF
		ELSE
			PowerState:=88;
		END_IF
	88:	(*All Done*)
		btn_PowerOn:=FALSE;
		PowerState:=0;
		Error:=FALSE;
		ErrorID:=0;
		Busy:=FALSE;
		InitDone:=TRUE;
		FB_power.On:=FALSE;
		fb_ton.IN:=FALSE;
		LED_Error:=FALSE;
	99:
		btn_PowerOn:=FALSE;
		PowerState:=99;
		Error:=TRUE;
		Busy:=FALSE;
		InitDone:=FALSE;
		FB_Power.On:=FALSE;
		fb_ton.IN:=FALSE;
		LED_Error:=TRUE;
END_CASE
END_ACTION

END_PROGRAM

// ---- POUs/1.CarrierMode/SingleCarrierMode/SingleCarrierMode.TcPOU
PROGRAM SingleCarrierMode
VAR_INPUT
		TopPositionNew:LREAL:=100;
	TopVelocityNew:LREAL:=0.5;
	btn_TopMove:BOOL;
	btn_TopStop:BOOL;
	BottomPositionNew:LREAL:=100;
	BottomVelocityNew:LREAL:=0.5;
	btn_BottomMove:BOOL;
	btn_BottomStop:BOOL;
	InPositionNew:LREAL:=100;
	InVelocityNew:LREAL:=0.5;
	btn_InMove:BOOL;
	btn_InStop:BOOL;
	OutPositionNew:LREAL:=100;
	OutVelocityNew:LREAL:=0.5;
	btn_OutMove:BOOL;
	btn_OutStop:BOOL;
END_VAR
VAR
	(*key Command*)

	(*Var*)
	fb_ton1:TON;
	fb_ton2:TON;
	fb_ton3:TON;
	fb_ton4:TON;
	fb_ton5:TON;
	fb_ton6:TON;
	(*Status*)
	State:DINT;
	Busy:BOOL;
	TopBusy:BOOL;
	BottomBusy:BOOL;
	InBusy:BOOL;
	OutBusy:BOOL;
	InitDone:BOOL;
	tm_state: DINT;
	ts_state: DINT;
	bm_state: DINT;
	bs_state: DINT;
	im_state: DINT;
	is_state: DINT;
	om_state: DINT;
	os_state: DINT;
	moni_State:DINT;
	(*PowerOff*)
	d_state: DINT;
	(*¼ì²âµ½ÏÞÎ»£¬»Ö¸´Move×´Ì¬*)
	FTrig_ReachLS: F_TRIG;
	FTrig_btn_GapMove: F_TRIG;
	InitPowerDone:BOOL;
	
END_VAR

TopPositionActual:=(Pos_LeftTopLin+Pos_RightTopLin)/2;
TopVelocityActual:=(Velo_LeftTopLin+Velo_RightTopLin)/2;
BottomPositionActual:=(Pos_LeftBottomLin+Pos_RightBOttomLin)/2;
BottomVelocityActual:=(Velo_LeftBottomLin+Velo_RightBOttomLin)/2;
InPositionActual:=(Pos_LeftInLin+Pos_RightInLin)/2;
InVelocityActual:=(Velo_LeftInLin+Velo_RightInLin)/2;
OutPositionActual:=(Pos_LeftOutLin+Pos_RightOutLin)/2;
OutVelocityActual:=(Velo_LeftOutLin+Velo_RightOutLin)/2;
(*btn_Power On/Off*)
IF btn_Power AND st_Power=0 THEN
	btn_PowerOn:=TRUE;
	btn_Power:=FALSE;
END_IF
IF btn_Power AND st_Power=1 THEN
	btn_PowerOff:=TRUE;
	btn_Power:=FALSE;
END_IF
IF btn_PowerOn THEN
	A_PowerOn();
END_IF
IF btn_PowerOff THEN
	A_PowerOff();
END_IF

(*************************Monitor All Carrirt Position*****************)
A_MonitoringAllAxis();
(*******************MOVE AND STOP*********************)
A_SingleCarrierMove();
A_SingleCarrierStop();
(**************ÏÞÎ»Åö´¥×´Ì¬»Ö¸´*******************************)
FTrig_ReachLS(CLK:=Unreach_LS_Far AND Unreach_LS_Near);
IF FTrig_ReachLS.Q THEN		(*FTrig_ReachLS.QÌ«¿ì£¬Ö»ÄÜÊ¹btn_TopStopÎªTRUE*)
	btn_TopStop:=TRUE;
	btn_BottomStop:=TRUE;
END_IF
IF btn_TopStop THEN			(*Òò´Ë£¬´Ë´¦Îªµ±Ö®Ç°btn_TopStopÎªTRUEÊ±£¬ÈËÎªÈÃbtn_BottomStopÎªTRUE*)
	btn_BottomStop:=TRUE;
END_IF

ACTION A_MonitoringAllAxis:
IF  st_Power<>0 THEN
		Diff_TopPos_actual:=Pos_leftTopLin-Pos_RightTopLin;
		Diff_TopVelo_actual:=Velo_leftTopLin-Velo_RightTopLin;
IF ABS(Pos_leftTopLin-Pos_RightTopLin)>Threshold_TopPos_SingleCarrier THEN
		btn_TopStop:=TRUE;
		btn_BottomStop:=TRUE;
		FB_PlcEmergencyStop();
		Error:=TRUE;
		ErrorID:=14;
		LED_Error:=TRUE;
ELSIF ABS(Velo_leftTopLin-Velo_RightTopLin)>Threshold_TopVelo_SingleCarrier  THEN
		(*btn_TopStop:=TRUE;
		btn_BottomStop:=TRUE;
		FB_PlcEmergencyStop();*)
		Error:=TRUE;
		ErrorID:=15;
(*Bottom Î»ÖÃºÍËÙ¶È±È¶Ô*)
ELSIF ABS(Pos_LeftBottomLin-Pos_RightBottomLin)>Threshold_BottomPos_SingleCarrier THEN
		btn_TopStop:=TRUE;
		btn_BottomStop:=TRUE;
		FB_PlcEmergencyStop();
		Error:=TRUE;
		ErrorID:=16;
		LED_Error:=TRUE;
ELSIF ABS(Velo_leftBottomLin-Velo_RightBottomLin)>Threshold_BottomVelo_SingleCarrier  THEN
		(*btn_TopStop:=TRUE;
		btn_BottomStop:=TRUE;
		FB_PlcEmergencyStop();*)
		Error:=TRUE;
		ErrorID:=17;
(*ÎÞLeftºÍRightËÙ¶ÈÎ»ÖÃµÄ¶Ô±È*)
END_IF
END_IF
IF  st_Power<>0 THEN
		Diff_InPos_actual:=Pos_leftInLin-Pos_RightInLin;
		Diff_InVelo_actual:=Velo_leftInLin-Velo_RightInLin;
IF ABS(Pos_leftInLin-Pos_RightInLin)>Threshold_InPos_SingleCarrier THEN
		btn_InStop:=TRUE;
		btn_OutStop:=TRUE;
		FB_PlcEmergencyStop();
		Error:=TRUE;
		ErrorID:=18;
		LED_Error:=TRUE;
ELSIF ABS(Velo_leftInLin-Velo_RightInLin)>Threshold_InVelo_SingleCarrier  THEN
		(*btn_InStop:=TRUE;
		btn_OutStop:=TRUE;
		FB_PlcEmergencyStop();*)
		Error:=TRUE;
		ErrorID:=19;
(*Out Î»ÖÃºÍËÙ¶È±È¶Ô*)
ELSIF ABS(Pos_LeftOutLin-Pos_RightOutLin)>Threshold_OutPos_SingleCarrier THEN
		btn_InStop:=TRUE;
		btn_OutStop:=TRUE;
		FB_PlcEmergencyStop();
		Error:=TRUE;
		ErrorID:=20;
		LED_Error:=TRUE;
ELSIF ABS(Velo_leftOutLin-Velo_RightOutLin)>Threshold_OutVelo_SingleCarrier  THEN
		(*btn_InStop:=TRUE;
		btn_OutStop:=TRUE;
		FB_PlcEmergencyStop();*)
		Error:=TRUE;
		ErrorID:=21;
(*ÎÞLeftºÍRightËÙ¶ÈÎ»ÖÃµÄ¶Ô±È*)
END_IF
END_IF
END_ACTION

ACTION A_PowerOff:
CASE d_state OF
		0:(*PowerOff*)
			FB_Power(Off:=TRUE);
				d_state:=1;
		1:
			IF NOT FB_power.OffStatus THEN
				d_state:=1;
			ELSE
				d_state:=88;
			END_IF
		88:(*ResetAllState*)
			btn_PowerOn:=FALSE;
			btn_TopMove:=FALSE;
			btn_TopStop:=FALSE;
			btn_BottomMove:=FALSE;
			btn_BottomStop:=FALSE;
			fb_ton1.IN:=FALSE;
			fb_ton2.IN:=FALSE;
			fb_ton3.IN:=FALSE;
			State:=0;
			Busy:=FALSE;
			InitPowerDone:=FALSE;
			Error:=FALSE;
			ErrorID:=0;
			tm_state:=0;
			ts_state:=0;
			bm_state:=0;
			bs_state:=0;
			btn_PowerOff:=FALSE;
			d_state:=0;
			Led_Run:=FALSE;
			Led_Error:=FALSE;
			moni_State:=0;
END_CASE
END_ACTION

ACTION A_PowerOn:
fb_ton3(PT:=T#0.5S);
CASE State OF
	0:	(*FB_Power_On*)
		FB_Power(On:=TRUE);
		fb_ton3.IN:=TRUE;
		State:=1;
	1:	(*wait*)
		FB_power();
		IF NOT FB_power.OnStatus THEN		(*FB_Power_OnÃ»ÓÐÖ´ÐÐÍê£¬wait£¬³¬Ê±FB Error*)
			IF NOT fb_ton3.Q THEN
				State:=1;
			ELSE
				ErrorID:=1;
				State:=99;
			END_IF
		ELSE
			State:=88;
		END_IF
	88:	(*All Done*)
		btn_PowerOn:=FALSE;
		State:=0;
		Error:=FALSE;
		ErrorID:=0;
		Busy:=FALSE;
		InitPowerDone:=TRUE;
		FB_power.On:=FALSE;
		fb_ton3.IN:=FALSE;
		LED_Error:=FALSE;
	99:
		Error:=TRUE;
		//ErrorID:=701;
		//ErrorDescription:='power on error';		
		btn_PowerOn:=FALSE;
		State:=99;
		Busy:=FALSE;
		InitPowerDone:=FALSE;
		fb_ton3.IN:=FALSE;
		LED_Error:=TRUE;
END_CASE
END_ACTION

ACTION A_SingleCarrierMove:
(*********************************************************************btn_TopMove*****************************************************************)
IF btn_TopMove THEN
		TopBusy:=TRUE;
		CASE tm_state OF
			0:
				FB_Move_Top.Mode:=1;						(*单梁模式*)
				FB_Move_Top.CoupleState:=st_Couple;			
				FB_Move_Top.PowerState:=st_Power;			
				FB_Move_Top.TopMove:=TRUE;				
				FB_Move_Top.TopPosition:=TopPositionNew;		
				FB_Move_Top.TopVelocity:=TopVelocityNew;		
				FB_Move_Top();								
				tm_state:=1;
			1:
				FB_Move_Top();
				LED_Run:=TRUE;
				IF NOT FB_Move_Top.TopDone THEN	
					tm_state:=1;
				ELSE					
					tm_state:=88;
				END_IF
			88:
				btn_TopMove:=FALSE;	
				LED_Run:=FALSE;
				tm_state:=0;
				TopBusy:=FALSE;
		END_CASE
END_IF

(*********************************************************************btn_BottomMove*****************************************************************)
IF btn_BottomMove THEN
		BottomBusy:=TRUE;
		CASE bm_state OF
			0:
				FB_Move_Bottom.Mode:=1;						
				FB_Move_Bottom.CoupleState:=st_Couple;			
				FB_Move_Bottom.PowerState:=st_Power;			
				FB_Move_Bottom.BottomMove:=TRUE;			
				FB_Move_Bottom.BottomPosition:=BottomPositionNew;		
				FB_Move_Bottom.BottomVelocity:=BottomVelocityNew;		
				FB_Move_Bottom();
				bm_state:=1;
			1:
				FB_Move_Bottom();
				IF NOT FB_Move_Bottom.BottomDone THEN
					LED_Run:=TRUE;
					bm_state:=1;
				ELSE
					bm_state:=88;
				END_IF
			88:
				BottomBusy:=FALSE;
				btn_TopMove:=FALSE;
				btn_BottomMove:=FALSE;
				bm_state:=0;
				LED_Run:=FALSE;
		END_CASE
END_IF
(*********************************************************************btn_TopMove*****************************************************************)
IF btn_InMove THEN
		InBusy:=TRUE;
		CASE im_state OF
			0:
				FB_Move_In.Mode:=1;						(*单梁模式*)
				FB_Move_In.CoupleState:=st_Couple;			
				FB_Move_In.PowerState:=st_Power;			
				FB_Move_In.InMove:=TRUE;				
				FB_Move_In.InPosition:=InPositionNew;		
				FB_Move_In.InVelocity:=InVelocityNew;		
				FB_Move_In();								
				im_state:=1;
			1:
				FB_Move_In();
				LED_Run:=TRUE;
				IF NOT FB_Move_In.InDone THEN	
					im_state:=1;
				ELSE					
					im_state:=88;
				END_IF
			88:
				btn_InMove:=FALSE;	
				LED_Run:=FALSE;
				im_state:=0;
				InBusy:=FALSE;
		END_CASE
END_IF

(*********************************************************************btn_BottomMove*****************************************************************)
IF btn_OutMove THEN
		OutBusy:=TRUE;
		CASE om_state OF
			0:
				FB_Move_Out.Mode:=1;						
				FB_Move_Out.CoupleState:=st_Couple;			
				FB_Move_Out.PowerState:=st_Power;			
				FB_Move_Out.OutMove:=TRUE;			
				FB_Move_Out.OutPosition:=OutPositionNew;		
				FB_Move_Out.OutVelocity:=OutVelocityNew;		
				FB_Move_Out();
				om_state:=1;
			1:
				FB_Move_Out();
				IF NOT FB_Move_Out.OutDone THEN
					LED_Run:=TRUE;
					om_state:=1;
				ELSE
					om_state:=88;
				END_IF
			88:
				OutBusy:=FALSE;
				btn_OutMove:=FALSE;
				om_state:=0;
				LED_Run:=FALSE;
		END_CASE
END_IF
END_ACTION

ACTION A_SingleCarrierStop:
(*******************************************************************btn_TopStop********************************************************************)

IF btn_TopStop THEN
	LED_Run:=FALSE;
	FB_Move_Top.TopReset:=TRUE;
	TopBusy:=FALSE;
	FB_Move_Top();
	btn_TopMove:=FALSE;	
	tm_state:=0;
	CASE ts_state OF
			0:
				FB_Stop_Top.Mode:=1;
				FB_Stop_Top.CoupleState:=st_Couple;
				FB_Stop_Top.PowerState:=st_Power;
				FB_Stop_Top.TopStop:=TRUE;	
				FB_Stop_Top();	
				ts_state:=1;
			1:
				FB_Stop_Top();
				IF NOT FB_Stop_Top.TopDone THEN
					ts_state:=1;
				ELSE
					ts_state:=88;
				END_IF
			88:
				btn_TopStop:=FALSE;	
				FB_Move_Top.TopReset:=FALSE;	
				ts_state:=0;
		END_CASE
END_IF
(*******************************************************************btn_BottomStop********************************************************************)
IF btn_BottomStop  THEN
	LED_Run:=FALSE;
	BottomMoveIndicator:=0;
	FB_Move_Bottom.BottomReset:=TRUE;
	BottomBusy:=FALSE;
	FB_Move_Bottom();			
	btn_BottomMove:=FALSE;			
	bm_state:=0;							
	CASE bs_state OF
			0:
				FB_Stop_Bottom.Mode:=1;							
				FB_Stop_Bottom.CoupleState:=st_Couple;			
				FB_Stop_Bottom.PowerState:=st_Power;			
				FB_Stop_Bottom.BottomStop:=TRUE;				
				FB_Stop_Bottom();								
				bs_state:=1;
			1:
				FB_Stop_Bottom();
				IF NOT FB_Stop_Bottom.BottomDone THEN		
					bs_state:=1;
				ELSE									
					bs_state:=88;
				END_IF
			88:
				btn_BottomStop:=FALSE;					
				FB_Move_Bottom.BottomReset:=FALSE;				
				bs_state:=0;
		END_CASE
END_IF
(*******************************************************************btn_InStop********************************************************************)

IF btn_InStop THEN
	LED_Run:=FALSE;
	FB_Move_In.InReset:=TRUE;
	InBusy:=FALSE;
	FB_Move_In();
	btn_InMove:=FALSE;	
	im_state:=0;
	CASE is_state OF
			0:
				FB_Stop_In.Mode:=1;
				FB_Stop_In.CoupleState:=st_Couple;
				FB_Stop_In.PowerState:=st_Power;
				FB_Stop_In.InStop:=TRUE;	
				FB_Stop_In();	
				is_state:=1;
			1:
				FB_Stop_In();
				IF NOT FB_Stop_In.InDone THEN
					is_state:=1;
				ELSE
					is_state:=88;
				END_IF
			88:
				btn_InStop:=FALSE;	
				FB_Move_In.InReset:=FALSE;	
				is_state:=0;
		END_CASE
END_IF
(*******************************************************************btn_OutStop********************************************************************)
IF btn_OutStop  THEN
	LED_Run:=FALSE;
	OutMoveIndicator:=0;
	FB_Move_Out.OutReset:=TRUE;
	OutBusy:=FALSE;
	FB_Move_Out();			
	btn_OutMove:=FALSE;			
	om_state:=0;							
	CASE os_state OF
			0:
				FB_Stop_Out.Mode:=1;							
				FB_Stop_Out.CoupleState:=st_Couple;			
				FB_Stop_Out.PowerState:=st_Power;			
				FB_Stop_Out.OutStop:=TRUE;				
				FB_Stop_Out();								
				os_state:=1;
			1:
				FB_Stop_Out();
				IF NOT FB_Stop_Out.OutDone THEN		
					os_state:=1;
				ELSE									
					os_state:=88;
				END_IF
			88:
				btn_OutStop:=FALSE;					
				FB_Move_Out.OutReset:=FALSE;				
				os_state:=0;
		END_CASE
END_IF
END_ACTION

END_PROGRAM

// ---- POUs/CommonFB/MainFB/FB_SetAxisPosition.TcPOU
(****************************************************************
NAME:			FB_SetAxisPosition
DATA:			2017.2.16
VERSION:		1.0.0
DESCRIPTION:	FB_SetAxisPosition
HISTORY:
				2017.2.16		NEW

***************************************************************)
FUNCTION_BLOCK FB_SetAxisPosition
VAR_INPUT
	//GapValueSet:LREAL:=0;
	ValueSet_LeftTop:LREAL:=0;
	ValueSet_RightTop:LREAL:=0;
	ValueSet_LeftBottom:LREAL:=0;
	ValueSet_RightBottom:LREAL:=0;
	ValueSet_LeftIn:LREAL:=0;
	ValueSet_RightIn:LREAL:=0;
	ValueSet_LeftOut:LREAL:=0;
	ValueSet_RightOut:LREAL:=0;
	Execute:BOOL;
END_VAR
VAR_OUTPUT
	FbID:DINT:=1001;
	State:DINT;
	Busy:BOOL;
	Done:BOOL;
	Error:BOOL;
	ErrorID:DINT;
END_VAR
VAR
	LeftTopLin_MC_SetPosition: MC_SetPosition;
	RightTopLin_MC_SetPosition: MC_SetPosition;
	LeftBottomLin_MC_SetPosition: MC_SetPosition;
	RightBottomLin_MC_SetPosition: MC_SetPosition;
	LeftInLin_MC_SetPosition: MC_SetPosition;
	RightInLin_MC_SetPosition: MC_SetPosition;
	LeftOutLin_MC_SetPosition: MC_SetPosition;
	RightOutLin_MC_SetPosition: MC_SetPosition;
	fb_ton: TON;
	FB_PlcEmergencyStop: FB_PlcEmergencyStop;

END_VAR

IF Execute THEN
Busy:=TRUE;
Done:=FALSE;
fb_ton(PT:=t#0.1s);
CASE State OF
	0:
		IF LeftTopLin_MC_SetPosition.Error OR RightTopLin_MC_SetPosition.Error
			OR LeftBottomLin_MC_SetPosition.Error OR RightBottomLin_MC_SetPosition.Error 
			OR LeftInLin_MC_SetPosition.Error OR RightInLin_MC_SetPosition.Error
			OR LeftOutLin_MC_SetPosition.Error OR RightOutLin_MC_SetPosition.Error THEN		(*FB Error*)
			ErrorID:=1;
			State:=99;
		ELSE
			State:=1;
		END_IF
	1:	(*Execute*)
		LeftTopLin_MC_SetPosition.Position:=ValueSet_LeftTop;
		LeftTopLin_MC_SetPosition.Execute:=TRUE;
		RightTopLin_MC_SetPosition.Position:=ValueSet_RightTop;
		RightTopLin_MC_SetPosition.Execute:=TRUE;
		LeftBottomLin_MC_SetPosition.Position:=ValueSet_LeftBottom;
		LeftBottomLin_MC_SetPosition.Execute:=TRUE;
		RightBottomLin_MC_SetPosition.Position:=ValueSet_RightBottom;
		RightBottomLin_MC_SetPosition.Execute:=TRUE;
		//
		LeftInLin_MC_SetPosition.Position:=ValueSet_LeftIn;
		LeftInLin_MC_SetPosition.Execute:=TRUE;
		RightInLin_MC_SetPosition.Position:=ValueSet_RightIn;
		RightInLin_MC_SetPosition.Execute:=TRUE;
		LeftOutLin_MC_SetPosition.Position:=ValueSet_LeftOut;
		LeftOutLin_MC_SetPosition.Execute:=TRUE;
		RightOutLin_MC_SetPosition.Position:=ValueSet_RightOut;
		RightOutLin_MC_SetPosition.Execute:=TRUE;
		A_SetPositionMC();
		fb_ton.IN:=TRUE;
		State:=2;
	2:	(*Wait*)
		A_SetPositionMC();
		IF NOT LeftTopLin_MC_SetPosition.Done OR NOT RightTopLin_MC_SetPosition.Done
			OR NOT LeftBottomLin_MC_SetPosition.Done OR NOT RightBottomLin_MC_SetPosition.Done 
			OR NOT LeftInLin_MC_SetPosition.Done OR NOT RightInLin_MC_SetPosition.Done
			OR NOT LeftOutLin_MC_SetPosition.Done OR NOT RightOutLin_MC_SetPosition.Done THEN		(*DoneÐÅºÅ²»µ½£¬¼ÌÐøµÈ´ý£¬Èç¹û³¬Ê±ÔòFB Error*)
			IF NOT fb_ton.Q THEN
				State:=2;
			ELSE
				ErrorID:=4;
				State:=99;
			END_IF
		ELSIF  LeftTopLin_MC_SetPosition.Done AND RightTopLin_MC_SetPosition.Done
			AND LeftBottomLin_MC_SetPosition.Done AND RightBottomLin_MC_SetPosition.Done 
			AND LeftInLin_MC_SetPosition.Done AND RightInLin_MC_SetPosition.Done
			AND LeftOutLin_MC_SetPosition.Done AND RightOutLin_MC_SetPosition.Done THEN		(*Done£¬×ªÏÂÒ»²½*)
			State:=88;
		ELSE
			ErrorID:=5;
			State:=99;
		END_IF
	88:
		Execute:=FALSE;
		State:=0;
		Busy:=FALSE;
		Done:=TRUE;
		Error:=FALSE;
		ErrorID:=0;
		LeftTopLin_MC_SetPosition.Execute:=FALSE;
		RightTopLin_MC_SetPosition.Execute:=FALSE;
		LeftBottomLin_MC_SetPosition.Execute:=FALSE;
		RightBottomLin_MC_SetPosition.Execute:=FALSE;
		LeftInLin_MC_SetPosition.Execute:=FALSE;
		RightInLin_MC_SetPosition.Execute:=FALSE;
		LeftOutLin_MC_SetPosition.Execute:=FALSE;
		RightOutLin_MC_SetPosition.Execute:=FALSE;
		fb_ton.IN:=FALSE;
	99:
		Execute:=FALSE;
		State:=99;
		Busy:=FALSE;
		Done:=FALSE;
		Error:=TRUE;
		LeftTopLin_MC_SetPosition.Execute:=FALSE;
		RightTopLin_MC_SetPosition.Execute:=FALSE;
		LeftBottomLin_MC_SetPosition.Execute:=FALSE;
		RightBottomLin_MC_SetPosition.Execute:=FALSE;
		LeftInLin_MC_SetPosition.Execute:=FALSE;
		RightInLin_MC_SetPosition.Execute:=FALSE;
		LeftOutLin_MC_SetPosition.Execute:=FALSE;
		RightOutLin_MC_SetPosition.Execute:=FALSE;
		fb_ton.IN:=FALSE;
	-100:
		FB_PlcEmergencyStop();
		Execute:=FALSE;
		State:=-100;
		Busy:=FALSE;
		Done:=FALSE;
		Error:=TRUE;
		LeftTopLin_MC_SetPosition.Execute:=FALSE;
		RightTopLin_MC_SetPosition.Execute:=FALSE;
		LeftBottomLin_MC_SetPosition.Execute:=FALSE;
		RightBottomLin_MC_SetPosition.Execute:=FALSE;
		
		LeftInLin_MC_SetPosition.Execute:=FALSE;
		RightInLin_MC_SetPosition.Execute:=FALSE;
		LeftOutLin_MC_SetPosition.Execute:=FALSE;
		RightOutLin_MC_SetPosition.Execute:=FALSE;
		fb_ton.IN:=FALSE;
END_CASE
END_IF

ACTION A_SetPositionMC:
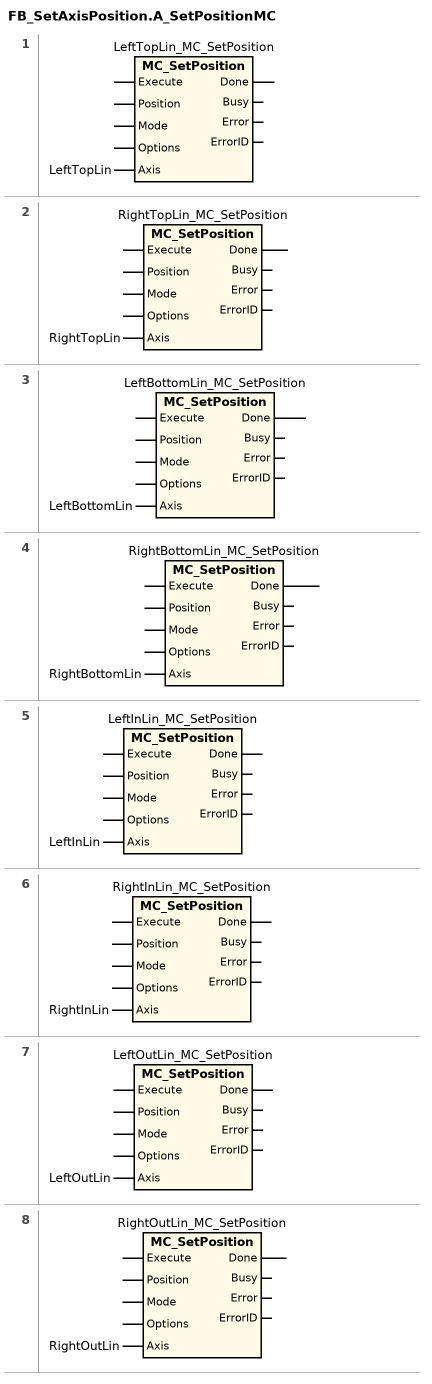
// NETWORK 1
LeftTopLin_MC_SetPosition(Axis := LeftTopLin); // MC_SetPosition

// NETWORK 2
RightTopLin_MC_SetPosition(Axis := RightTopLin); // MC_SetPosition

// NETWORK 3
LeftBottomLin_MC_SetPosition(Axis := LeftBottomLin); // MC_SetPosition

// NETWORK 4
RightBottomLin_MC_SetPosition(Axis := RightBottomLin); // MC_SetPosition

// NETWORK 5
LeftInLin_MC_SetPosition(Axis := LeftInLin); // MC_SetPosition

// NETWORK 6
RightInLin_MC_SetPosition(Axis := RightInLin); // MC_SetPosition

// NETWORK 7
LeftOutLin_MC_SetPosition(Axis := LeftOutLin); // MC_SetPosition

// NETWORK 8
RightOutLin_MC_SetPosition(Axis := RightOutLin); // MC_SetPosition
END_ACTION

END_FUNCTION_BLOCK

// ---- POUs/CommonFB/MainFB/FB_SetMotorAxisPosition.TcPOU
(****************************************************************
NAME:			FB_SetAxisPosition
DATA:			2017.2.16
VERSION:		1.0.0
DESCRIPTION:	FB_SetAxisPosition
HISTORY:
				2017.2.16		NEW

***************************************************************)
FUNCTION_BLOCK FB_SetMotorAxisPosition
VAR_INPUT
	//GapValueSet:LREAL:=0;
	ValueSet_LeftTop:LREAL:=0;
	ValueSet_RightTop:LREAL:=0;
	ValueSet_LeftBottom:LREAL:=0;
	ValueSet_RightBottom:LREAL:=0;
	ValueSet_LeftIn:LREAL:=0;
	ValueSet_RightIn:LREAL:=0;
	ValueSet_LeftOut:LREAL:=0;
	ValueSet_RightOut:LREAL:=0;
	Execute:BOOL;
END_VAR
VAR_OUTPUT
	FbID:DINT:=1001;
	State:DINT;
	Busy:BOOL;
	Done:BOOL;
	Error:BOOL;
	ErrorID:DINT;
END_VAR
VAR
	LeftTopMotor_MC_SetPosition: MC_SetPosition;
	RightTopMotor_MC_SetPosition: MC_SetPosition;
	LeftBottomMotor_MC_SetPosition: MC_SetPosition;
	RightBottomMotor_MC_SetPosition: MC_SetPosition;
	LeftInMotor_MC_SetPosition: MC_SetPosition;
	RightInMotor_MC_SetPosition: MC_SetPosition;
	LeftOutMotor_MC_SetPosition: MC_SetPosition;
	RightOutMotor_MC_SetPosition: MC_SetPosition;
	fb_ton: TON;
	FB_PlcEmergencyStop: FB_PlcEmergencyStop;

END_VAR

IF Execute THEN
Busy:=TRUE;
Done:=FALSE;
fb_ton(PT:=t#0.1s);
CASE State OF
	0:
		IF LeftTopMotor_MC_SetPosition.Error OR RightTopMotor_MC_SetPosition.Error
			OR LeftBottomMotor_MC_SetPosition.Error OR RightBottomMotor_MC_SetPosition.Error 
			OR LeftInMotor_MC_SetPosition.Error OR RightInMotor_MC_SetPosition.Error
			OR LeftOutMotor_MC_SetPosition.Error OR RightOutMotor_MC_SetPosition.Error THEN		(*FB Error*)
			ErrorID:=1;
			State:=99;
		ELSE
			State:=1;
		END_IF
	1:	(*Execute*)
		LeftTopMotor_MC_SetPosition.Position:=ValueSet_LeftTop;
		LeftTopMotor_MC_SetPosition.Execute:=TRUE;
		RightTopMotor_MC_SetPosition.Position:=ValueSet_RightTop;
		RightTopMotor_MC_SetPosition.Execute:=TRUE;
		LeftBottomMotor_MC_SetPosition.Position:=ValueSet_LeftBottom;
		LeftBottomMotor_MC_SetPosition.Execute:=TRUE;
		RightBottomMotor_MC_SetPosition.Position:=ValueSet_RightBottom;
		RightBottomMotor_MC_SetPosition.Execute:=TRUE;
		//
		LeftInMotor_MC_SetPosition.Position:=ValueSet_LeftIn;
		LeftInMotor_MC_SetPosition.Execute:=TRUE;
		RightInMotor_MC_SetPosition.Position:=ValueSet_RightIn;
		RightInMotor_MC_SetPosition.Execute:=TRUE;
		LeftOutMotor_MC_SetPosition.Position:=ValueSet_LeftOut;
		LeftOutMotor_MC_SetPosition.Execute:=TRUE;
		RightOutMotor_MC_SetPosition.Position:=ValueSet_RightOut;
		RightOutMotor_MC_SetPosition.Execute:=TRUE;
		A_SetPositionMC();
		fb_ton.IN:=TRUE;
		State:=2;
	2:	(*Wait*)
		A_SetPositionMC();
		IF NOT LeftTopMotor_MC_SetPosition.Done OR NOT RightTopMotor_MC_SetPosition.Done
			OR NOT LeftBottomMotor_MC_SetPosition.Done OR NOT RightBottomMotor_MC_SetPosition.Done 
			OR NOT LeftInMotor_MC_SetPosition.Done OR NOT RightInMotor_MC_SetPosition.Done
			OR NOT LeftOutMotor_MC_SetPosition.Done OR NOT RightOutMotor_MC_SetPosition.Done THEN		(*DoneÐÅºÅ²»µ½£¬¼ÌÐøµÈ´ý£¬Èç¹û³¬Ê±ÔòFB Error*)
			IF NOT fb_ton.Q THEN
				State:=2;
			ELSE
				ErrorID:=4;
				State:=99;
			END_IF
		ELSIF  LeftTopMotor_MC_SetPosition.Done AND RightTopMotor_MC_SetPosition.Done
			AND LeftBottomMotor_MC_SetPosition.Done AND RightBottomMotor_MC_SetPosition.Done 
			AND LeftInMotor_MC_SetPosition.Done AND RightInMotor_MC_SetPosition.Done
			AND LeftOutMotor_MC_SetPosition.Done AND RightOutMotor_MC_SetPosition.Done THEN		(*Done£¬×ªÏÂÒ»²½*)
			State:=88;
		ELSE
			ErrorID:=5;
			State:=99;
		END_IF
	88:
		Execute:=FALSE;
		State:=0;
		Busy:=FALSE;
		Done:=TRUE;
		Error:=FALSE;
		ErrorID:=0;
		LeftTopMotor_MC_SetPosition.Execute:=FALSE;
		RightTopMotor_MC_SetPosition.Execute:=FALSE;
		LeftBottomMotor_MC_SetPosition.Execute:=FALSE;
		RightBottomMotor_MC_SetPosition.Execute:=FALSE;
		LeftInMotor_MC_SetPosition.Execute:=FALSE;
		RightInMotor_MC_SetPosition.Execute:=FALSE;
		LeftOutMotor_MC_SetPosition.Execute:=FALSE;
		RightOutMotor_MC_SetPosition.Execute:=FALSE;
		fb_ton.IN:=FALSE;
	99:
		Execute:=FALSE;
		State:=99;
		Busy:=FALSE;
		Done:=FALSE;
		Error:=TRUE;
		LeftTopMotor_MC_SetPosition.Execute:=FALSE;
		RightTopMotor_MC_SetPosition.Execute:=FALSE;
		LeftBottomMotor_MC_SetPosition.Execute:=FALSE;
		RightBottomMotor_MC_SetPosition.Execute:=FALSE;
		LeftInMotor_MC_SetPosition.Execute:=FALSE;
		RightInMotor_MC_SetPosition.Execute:=FALSE;
		LeftOutMotor_MC_SetPosition.Execute:=FALSE;
		RightOutMotor_MC_SetPosition.Execute:=FALSE;
		fb_ton.IN:=FALSE;
	-100:
		FB_PlcEmergencyStop();
		Execute:=FALSE;
		State:=-100;
		Busy:=FALSE;
		Done:=FALSE;
		Error:=TRUE;
		LeftTopMotor_MC_SetPosition.Execute:=FALSE;
		RightTopMotor_MC_SetPosition.Execute:=FALSE;
		LeftBottomMotor_MC_SetPosition.Execute:=FALSE;
		RightBottomMotor_MC_SetPosition.Execute:=FALSE;
		
		LeftInMotor_MC_SetPosition.Execute:=FALSE;
		RightInMotor_MC_SetPosition.Execute:=FALSE;
		LeftOutMotor_MC_SetPosition.Execute:=FALSE;
		RightOutMotor_MC_SetPosition.Execute:=FALSE;
		fb_ton.IN:=FALSE;
END_CASE
END_IF

ACTION A_SetPositionMC:
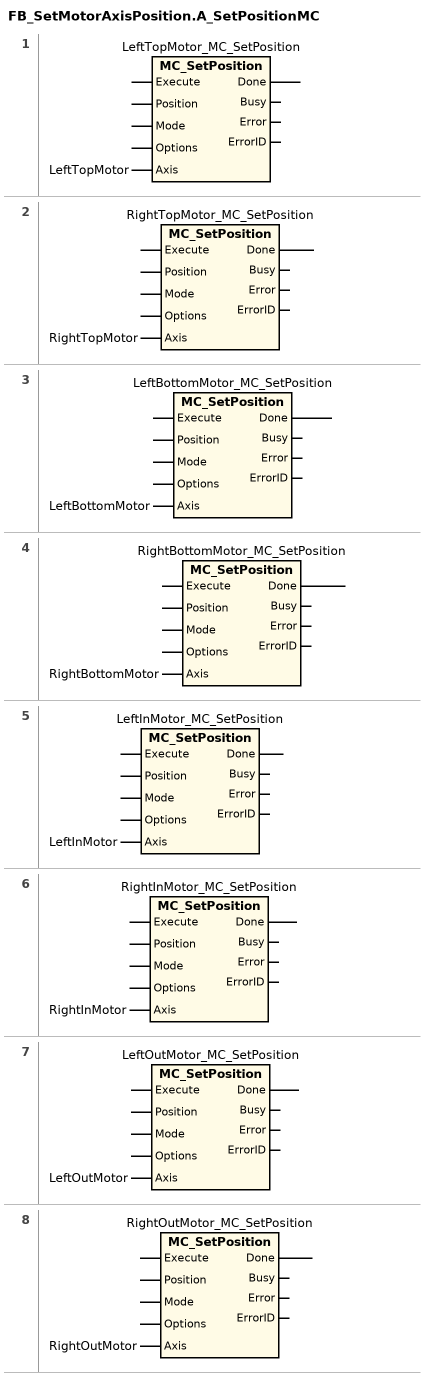
// NETWORK 1
LeftTopMotor_MC_SetPosition(Axis := LeftTopMotor); // MC_SetPosition

// NETWORK 2
RightTopMotor_MC_SetPosition(Axis := RightTopMotor); // MC_SetPosition

// NETWORK 3
LeftBottomMotor_MC_SetPosition(Axis := LeftBottomMotor); // MC_SetPosition

// NETWORK 4
RightBottomMotor_MC_SetPosition(Axis := RightBottomMotor); // MC_SetPosition

// NETWORK 5
LeftInMotor_MC_SetPosition(Axis := LeftInMotor); // MC_SetPosition

// NETWORK 6
RightInMotor_MC_SetPosition(Axis := RightInMotor); // MC_SetPosition

// NETWORK 7
LeftOutMotor_MC_SetPosition(Axis := LeftOutMotor); // MC_SetPosition

// NETWORK 8
RightOutMotor_MC_SetPosition(Axis := RightOutMotor); // MC_SetPosition
END_ACTION

END_FUNCTION_BLOCK

// ---- POUs/MAIN.TcPOU
PROGRAM MAIN
VAR
	pbSingleCarrierMode: BOOL:=FALSE;
	pbDebugMode:BOOL:=FALSE;
	fb_led_Show: FB_LedShow;
	btn_reset: BOOL;
	CPMU_PLC_Reset: PLC_Reset;
	d_state: DINT;
	CPMU_PLC_Start: PLC_Start;
	powerStatus:BOOL;

(*TwinSAFE*)
	Safe_run AT%Q*:BOOL;
	Err_Ack AT %Q*:BOOL;
	Estop_RunAndRestart AT %Q*:BOOL;
	AX5805_Error_Ack AT %Q*:BOOL;
	Led_Run  AT %Q*:BOOL;
	Led_Error  AT %Q*:BOOL;

	FB_ERROR AT%I*:BOOL;
	COM_ERROR AT%I*:BOOL;
	//OUT_ERROR AT%I*:BOOL;
	Estop_Out AT%I*:BOOL;

	SafeStatus:INT;
	SafePLCRunOK: BOOL;
	fb_ton: TON;
	fb_ton2: TON;
	fb_ton3: TON;
	fb_ton1: TON;
	fb_ton0: TON;
(*IO*)
	el1808_D1  AT%I* :ARRAY[1..16] OF BOOL;
	EStopTrig:BOOL;
(*setAxisPosition*)
	SetAxisPosState: INT;
	FB_Set_AxisPosition:FB_SetAxisPosition;
	fb_ton4: TON;
	fb_ton5: TON;
	fb_ton6: TON;
	SerAxisPositionDone: BOOL;

	i: INT;
	j: INT;

(****RS232***)
	fbEL6001	: FB_SerialCom;


(*Torque*)
	Torque_LT AT%I*:INT;
	Torque_RT AT%I*:INT;
	Torque_LB AT%I*:INT;
	Torque_RB AT%I*:INT;
	Torque_LI AT%I*:INT;
	Torque_RI AT%I*:INT;
	Torque_LO AT%I*:INT;
	Torque_RO AT%I*:INT;
(**)
	btn_setAxisPosition: BOOL;
	ValueSet_LeftTop:LREAL;
	ValueSet_RightTop:LREAL;
	ValueSet_LeftBottom:LREAL;
	ValueSet_RightBottom:LREAL;
	ValueSet_LeftIn:LREAL;
	ValueSet_RightIn:LREAL;
	ValueSet_LeftOut:LREAL;
	ValueSet_RightOut:LREAL;
(**)
	RestartTC: TC_Restart;
	
(*recipe*)
	RecipeINT:INT;
	RecipeBOOL:BOOL;
	RecipeManCommands: RecipeManCommands;
	SaveParameter : BOOL;  //保存文件
	LoadParameter : BOOL;  //读取文件
	Save_R_TRIG   : R_TRIG;
	Read_R_TRIG   : R_TRIG;
	loadparameterStatus: INT;
	RecipeBOOL2:BOOL;
	ReturnDwordLoad: DWORD;
	InsertionDeviceName:STRING;
(*UserMode*)
	pbUserMode: BOOL:=TRUE;
	EL1904 AT%I* :ARRAY[1..48] OF BOOL;
	setAxisPositionEnable: BOOL;
	state_loadParameters: INT;
	state_setLEPosBias: INT;
	//
	PositionBiasSet:BOOL;
	MC_SetLEPosBias_LeftTop:MC_WriteParameter;
	MC_SetLEPosBias_RightTop:MC_WriteParameter;
	MC_SetLEPosBias_LeftBottom:MC_WriteParameter;
	MC_SetLEPosBias_RightBottom:MC_WriteParameter;
	MC_SetLEPosBias_LeftIn:MC_WriteParameter;
	MC_SetLEPosBias_RightIn:MC_WriteParameter;
	MC_SetLEPosBias_LeftOut:MC_WriteParameter;
	MC_SetLEPosBias_RightOut:MC_WriteParameter;
	PositionBias_LeftTop: LREAL:=0;
	PositionBias_RightTop: LREAL:=0;
	PositionBias_LeftBottom: LREAL:=0;
	PositionBias_RightBottom: LREAL:=0;
	PositionBias_LeftIn: LREAL:=0;
	PositionBias_RightIn: LREAL:=0;
	PositionBias_LeftOut: LREAL:=0;
	PositionBias_RightOut: LREAL:=0;

	LoadLEPB_R_TRIG: R_TRIG;
	PositionBiasTON: TON;
	
	//
	OPC_TEST_Bi:BOOL:=TRUE; (*~ (OPC:1:available for OPC Clients) *)
	OPC_TEST_Bi2:BOOL;(*~ (OPC:1:available for OPC Clients) *)
	//
	HasTemperatureSensorOrNot:BOOL;//Only IVU or CPMU
	(*Sensor Reading*)
	Sensor_Reading_1 AT %I*:ARRAY[0..3] OF BYTE;
	Sensor_Reading_2 AT %I*:ARRAY[0..3] OF BYTE;
	Sensor_Reading_3 AT %I*:ARRAY[0..3] OF BYTE;
	Sensor_Reading_4 AT %I*:ARRAY[0..3] OF BYTE;
	Sensor_Reading_5 AT %I*:ARRAY[0..3] OF BYTE;
	Sensor_Reading_6 AT %I*:ARRAY[0..3] OF BYTE;
	Sensor_Reading_7 AT %I*:ARRAY[0..3] OF BYTE;
	Sensor_Reading_8 AT %I*:ARRAY[0..3] OF BYTE;
	Sensor_Reading_DpState AT %I*:USINT;
	Sensor_Reading_ExtDiagFlag AT %I*:BOOL;
	TemperatureSensors_1:LREAL;
	TemperatureSensors_2:LREAL;
	TemperatureSensors_3:LREAL;
	TemperatureSensors_4:LREAL;
	TemperatureSensors_5:LREAL;
	TemperatureSensors_6:LREAL;
	TemperatureSensors_7:LREAL;
	TemperatureSensors_8:LREAL;
	dut_sensor_datas_1:DUT_SENSOR_DATAS_1;
	dut_sensor_datas_2:DUT_SENSOR_DATAS_2;
	dut_sensor_datas_3:DUT_SENSOR_DATAS_3;
	dut_sensor_datas_4:DUT_SENSOR_DATAS_4;
	dut_sensor_datas_5:DUT_SENSOR_DATAS_5;
	dut_sensor_datas_6:DUT_SENSOR_DATAS_6;
	dut_sensor_datas_7:DUT_SENSOR_DATAS_7;
	dut_sensor_datas_8:DUT_SENSOR_DATAS_8;
	//
	temperature_gradient_2_To_1:LREAL;
	temperature_gradient_3_To_2:LREAL;
	temperature_gradient_5_To_4:LREAL;
	temperature_gradient_6_To_5:LREAL;
	temperature_gradient_max:LREAL;
	//
	temperature_average:LREAL;
	A_SetLinearEncoderPositionBias_Enable: BOOL;
	
		//
	temperatureStatus:INT;//0：有传感器度数错误；1:常温；2:低温；3:常温和低温中间态
	CryogenicTemperatureThreshold:LREAL:=80;//80K以下归划分为低温
	RoomTemperatureThreshold:LREAL:=293;//293K以上划分为常温
	//CPMU cryogenix ON/FF
	CryogenicCompensationOn:BOOL;
	CryogenicCompensationConditionsReady:BOOL;
	CryogenicCompensation_LeftTop:LREAL;
	CryogenicCompensation_RightTop:LREAL;
	CryogenicCompensation_LeftBottom:LREAL;
	CryogenicCompensation_RightBottom:LREAL;
	CryogenicCompensationDone: BOOL;
	
